fb_WormWeight(
	nLine:= 1, 
	UnitID:= 5, 
	fFast_Speed_vibrating_funnel:= fFast_Speed_vibrating_funnel, 
	fSlow_Speed_vibrating_funnel_1:= fSlow_Speed_vibrating_funnel_1, 
	fSlow_Speed_vibrating_funnel_2:= fSlow_Speed_vibrating_funnel_2, 
	fDerisedWeight_Worm:= fDerisedWeight_Worm, 
	fChangeMode_Worm_1:= fChangeMode_Worm_1, 
	fChangeMode_Worm_2:= fChangeMode_Worm_2, 
	fMaxWeight_Worm:= fMaxWeight_Worm, 
	fPerStop_Worm:= fPerStop_Worm, 
	fTimer_Worm:= fTimer_Worm, 
	fTimer_Alarm_Worm:= fTimer_Alarm_Worm, 
	fTimer_Check_Worm:= fTimer_Check_Worm, 
	fTimer_Check_Cylinder:= fTimer_Check_Cylinder, 
	fDelta_Worm:= fDelta_Worm,
	fTimer_Error_Worm:= fTimer_Error_Worm, 
	fProductLog=> fProductLog[2],
	bStatus_Worm=>bStatus_Worm,
	Time_start=>Time_Start_Worm_line1,
	Time_Stop=>Time_Stop_Worm_line1,
	status=>bStatus_Worm_line1,
	fweight_iot =>fWeight_Worm_line1);

IF bClear1 THEN
	nResult_false1 := 0;
	nResult_true1 := 0;
	nCount1 := 0;
	bClear1 := FALSE;
END_IF	

fDerisedWeight_Food_line1	:= fDerisedWeight_Food;
fDerisedWeight_Worm_line1	:= fDerisedWeight_Worm;
fActDelta_Food_line1		:= fb_FoodWeight.fActDelta_Food;
fActDelta_Worm_line1		:= fb_WormWeight.fActDelta_Worm;
fDelta_Food_line1			:= fb_FoodWeight.fDelta_Food;
fDelta_Worm_line1			:= fb_WormWeight.fDelta_Worm;
	
IF getuser = 'Operator' THEN
	bypassfood := FALSE;
	bypassWorm := FALSE;
END_IF

ACTION Auto:
CASE nState OF
	0:// int
		bStatus_Food_order[1] := FALSE;
		bStatus_Worm_order[1] := FALSE;
		bStatus_Lid_order[1]  := FALSE;
		fb_Transfer.Init();
		fb_FoodWeight.SetZero();
		fb_WormWeight.SetZero();
		nDoneTransferStop	  := 0;
		i1 		:= 0;
		i2 		:= 0;
		i3 		:= 0;
		bfinish1	:= TRUE;
		nState 	:= 1;
		
	1: // Start
		nState_FoodWeight := 0;
		nState_WormWeight := 0;
		nState_LidSupply := 0;
		nState_LidClose := 0;
		bResetAuto1			:= FALSE;
		bDoneCupSupply 		:= FALSE;
		bDoneFoodWeight 	:= FALSE;
		bDoneWormWeight 	:= FALSE;
		bDoneLidSupply 		:= FALSE;
		bDoneLidClose 		:= FALSE;
		fb_FoodWeight.SetZero();
		fb_WormWeight.SetZero();
		nState := 11;
	11:
		bResetAuto1			:= FALSE;
		nState_Dropcup := 0;
		nState_Transfer := 0;
		bStop1 := FALSE;
		bShift_is_over1 := FALSE;
		bStatusStart1 := FALSE;
		fb_FoodMixer.Stop();
		nStatus1	:= 'STOP';
		bFinishCupSupply 	:= FALSE;
		bFinishFoodWeight 	:= FALSE;
		bFinishWormWeight	:= FALSE;
		bFinishLidSupply	:= FALSE;
		bFinishLidClose		:= FALSE;
		bFinishTransfer		:= FALSE;
		bfinish1	:= TRUE;
		nState := 22;
	22:
		IF bStart1 THEN
			bfinish1		:= FALSE;
			bStatusStart1 	:= TRUE;
			bToDropcup1 	:= FALSE;
			bResetAuto1		:= TRUE;
			status			:= 'RUN';
			nState := 2;
		END_IF
		
	2: // start mode auto
		bfinish1		:= FALSE;
		nStatus1	:= 'RUN';
		bResetAuto1		:= TRUE;
		bStart1 := FALSE;
		IF bypassfood THEN
			fb_FoodMixer.Stop();
		ELSE
			fb_FoodMixer.Auto();
		END_IF
		fb_CupSupply.CheckCup();
		fb_LidSupply.CheckLid();
		bDone(CLK := bDoneTransfer);
		CASE nstateCycle OF 
			0:
				fbTimerCycle(IN := TRUE, PT := T#100S);
				IF bDone.Q THEN
					nstateCycle := 1;
				END_IF
			1:
				timeCycle := TIME_TO_REAL(fbTimerCycle.ET)/1000;
				nstateCycle := 2;
			2: 
				fproduct :=  REAL_TO_INT(3600/(timeCycle+0.001));
				fbTimerCycle(IN := FALSE);
				nstateCycle := 0;
		END_CASE
		CASE nState_Dropcup OF
			0:// waiting for transfer
				fbDelay(IN := FALSE);
				fb_CupSupply.HoldCup();
				IF bToDropcup1 THEN
					nState_Dropcup := 1;
				END_IF
			1:// dropcup
				IF fb_CupSupply.DropCup() THEN
					bDoneCupSupply := TRUE;
					bToDropcup1 := FALSE;
					nState_Dropcup := 2;
				END_IF
			2:
				fbDelay(IN := TRUE, PT := T#300MS);
				IF fbDelay.Q THEN
					nState_Dropcup := 0;
				END_IF
		END_CASE
		
		CASE nState_FoodWeight OF
			0:// waiting for transfer
				IF bDoneTransfer THEN
					i1 := i1 + 1;
					fbTimer(IN := FALSE);
					nState_FoodWeight := 1;	
				END_IF
			1:// Check cup present
				IF NOT fb_FoodWeight.bIsCupPresent THEN
					IF bypassfood THEN
						nState_FoodWeight := 3;
						bStatus_Food_order[i1] := TRUE;
					ELSE
						nState_FoodWeight := 2;
					END_IF
				ELSE
					bStatus_Food_order[i1] := FALSE;
					nState_FoodWeight := 3;
				END_IF
			2:// FoodWeight
				IF NOT fb_FoodWeight.bIsCupPresent THEN
					IF fb_FoodWeight.Auto() THEN
						bStatus_Food_order[i1] := bStatus_Food;
						nState_FoodWeight := 3;
					END_IF
				ELSE
					nState_FoodWeight := 22;
				END_IF 
			22:
				fbTimer(IN := TRUE, PT := T#0.3S);
				fb_FoodWeight.Auto();
				IF fbTimer.Q THEN
					fb_FoodWeight.Init();
					nState_FoodWeight := 0;
				END_IF
			3:// check i
				IF i1 < 3 THEN
					nState_FoodWeight := 5;
				ELSE 
					i1 := 2;
					nState_FoodWeight := 4;
				END_IF
			4:// dao vi tri
				bStatus_Food_order[1] := bStatus_Food_order[2];
				bStatus_Food_order[2] := bStatus_Food_order[3];
				nState_FoodWeight := 5;
			5:// Done
				bDoneFoodWeight := TRUE;
				nState_FoodWeight := 10;
		END_CASE
		
		CASE nState_WormWeight OF
			0: // waiting for transfer
				IF bDoneTransfer THEN
					i2 := i2 + 1;;
					fbTimer(IN := FALSE);
					nState_WormWeight := 1;
				END_IF
			1:
				IF NOT fb_WormWeight.bIsCupPresent THEN
					nCount1 := nCount1 + 1;
					nState_WormWeight := 11;
				ELSE
					bStatus_Worm_order[i2] := FALSE;
					nState_WormWeight := 3;
				END_IF
			11: // check food
				IF bStatus_Food_order[1] THEN
					IF bypassWorm THEN
						nState_WormWeight := 3;
						bStatus_Worm_order[i2] := TRUE;
					ELSE
						nState_WormWeight := 2;
					END_IF
				ELSE
					bStatus_Worm_order[i2] := FALSE;
					nState_WormWeight := 3;
				END_IF	
			2:// WormWeight
				IF NOT fb_WormWeight.bIsCupPresent THEN
					IF fb_WormWeight.Auto() THEN
						bStatus_Worm_order[i2] := bStatus_Worm;
						nState_WormWeight := 3;
					END_IF
				ELSE
					nState_WormWeight := 22;
				END_IF
			22:
				fbTimer(IN := TRUE, PT := T#0.3S);
				fb_WormWeight.Auto(); 
				IF fbTimer.Q THEN
					fb_WormWeight.Init();
					nState_WormWeight := 0;
				END_IF
			3:// check i
				IF bStatus_Worm_order[i2] THEN
					nResult_true1 := nResult_true1 + 1;
				END_IF
				IF i2 < 3 THEN
					nState_WormWeight := 5;
				ELSE
					i2 := 2;
					nState_WormWeight := 4;
				END_IF
			4:// dao vi tri
				nResult_false1 := nCount1 - nResult_true1;
				bStatus_Worm_order[1] := bStatus_Worm_order[2];
				bStatus_Worm_order[2] := bStatus_Worm_order[3];
				nState_WormWeight 	  := 5;
			5:// Done 
				bDoneWormWeight       := TRUE;
				nState_WormWeight	  := 10;
		END_CASE
		
		CASE nState_LidSupply OF
			0:// waiting for transfer
				IF bDoneTransfer THEN
					i3 := i3 + 1;
					nState_LidSupply := 1;
				END_IF
			1:// check worm
				IF bStatus_Worm_order[1] THEN
					IF bypassLid THEN
						bStatus_Lid_order[i3] := FALSE;
						nState_LidSupply := 4;
					ELSE
						nState_LidSupply := 2;
					END_IF
				ELSE
					bStatus_Lid_order[i3] := FALSE;
					nState_LidSupply := 4;
				END_IF
			2:// take lid
				IF fb_LidSupply.TakeLid() THEN
					nState_LidSupply := 3;
				END_IF
			3:// drop lid
				IF fb_LidSupply.DropLid() THEN
					bStatus_Lid_order[i3] := TRUE;
					nState_LidSupply := 4;
				END_IF
			4:// check i
				IF i3 < 3 THEN
					nState_LidSupply := 6;
				ELSE
					i3 := 2;
					nState_LidSupply := 5;
				END_IF
			5:// dao vi tri
				bStatus_Lid_order[1] := bStatus_Lid_order[2];
				bStatus_Lid_order[2] := bStatus_Lid_order[3];
				nState_LidSupply 	 := 6;
			6:// Done
				bDoneLidSupply 		 := TRUE;
				nState_LidSupply 	 := 10;
		END_CASE
		
		CASE nState_LidClose OF
			0: // waiting for transfer
				IF bDoneTransfer THEN
					nState_LidClose := 1;
				END_IF
			1:// Check lid supply
				IF  bStatus_Lid_order[1] THEN
					nState_LidClose := 2;
				ELSE
					nState_LidClose := 3;
				END_IF
			2:// Close lid
				IF fb_LidClose.CloseLid() THEN
					nState_LidClose := 3;
				END_IF
			3://Done
				bDoneLidClose := TRUE;
				nState_LidClose := 10;
		END_CASE
		
		CASE nState_Transfer OF
			0:// waiting for Done module
				IF nDoneTransfer = 0 THEN
					nState_Transfer := 1;
				ELSIF nDoneTransfer > 0 THEN
					IF bDoneCupSupply AND bDoneFoodWeight AND bDoneWormWeight AND bDoneLidSupply AND bDoneLidClose THEN
						nState_Transfer := 1;
					END_IF
				END_IF
			1:
				IF fb_CupSupply.isCupDrop THEN
					bDoneCupSupply 	:= FALSE;
					bDoneFoodWeight := FALSE;
					bDoneWormWeight := FALSE;
					bDoneLidSupply 	:= FALSE;
					bDoneLidClose 	:= FALSE;
					nState_Transfer := 11;
				ELSE 
					F_SetError(2,nLine:=1);
				END_IF
			11:// transfer
				IF fb_Transfer.Auto() THEN
					nShoot1 := nShoot1 + 1; 
					nState_Transfer:= 2;
				END_IF
			2:
				nState_FoodWeight := 0;
				nState_WormWeight := 0;
				nState_LidSupply  := 0;
				nState_LidClose	  := 0;
				nState_Transfer	  := 0;
		END_CASE
		//Stop button
		IF bStop1 THEN
			nState := 3;
			bStartLine1 := FALSE;
		ELSIF bShift_is_over1 THEN
			nState := 4;
		END_IF
	3://Stop
		bfinish1 := FALSE;
		fb_CupSupply.CheckCup();
		fb_LidSupply.CheckLid();
		bResetAuto1		:= TRUE;
		nStatus1	:= 'RUN';
		IF bypassfood THEN
			fb_FoodMixer.Stop();
		ELSE
			fb_FoodMixer.Auto();
		END_IF
		CASE nState_Dropcup OF
			0:// waiting for transfer
				fbDelay(IN := FALSE);
				fb_CupSupply.HoldCup();
				IF bToDropcup1 THEN
					nState_Dropcup := 1;
				END_IF
				IF bFinishTransfer THEN
					nState_Dropcup := 10;
				END_IF
			1:// dropcup
				IF fb_CupSupply.DropCup() THEN
					bDoneCupSupply := TRUE;
					bToDropcup1 := FALSE;
					nState_Dropcup := 2;
				END_IF
			2:
				fbDelay(IN := TRUE, PT := T#300MS);
				IF fbDelay.Q THEN
					nState_Dropcup := 10;
				END_IF
			10:// finish
				bDoneCupSupply := TRUE;
				bFinishCupSupply := TRUE;
		END_CASE
		
		CASE nState_FoodWeight OF
			0:// waiting for transfer
				IF bDoneTransfer THEN
					i1 := i1 + 1;
					fbTimer(IN := FALSE);
					nState_FoodWeight := 1;	
				END_IF
			1:// Check cup present
				IF NOT fb_FoodWeight.bIsCupPresent THEN
					IF bypassfood THEN
						nState_FoodWeight := 3;
						bStatus_Food_order[i1] := TRUE;
					ELSE
						nState_FoodWeight := 2;
					END_IF
				ELSE
					bStatus_Food_order[i1] := FALSE;
					nState_FoodWeight := 3;
				END_IF
			2:// FoodWeight
				IF NOT fb_FoodWeight.bIsCupPresent THEN
					IF fb_FoodWeight.Auto() THEN
						bStatus_Food_order[i1] := bStatus_Food;
						nState_FoodWeight := 3;
					END_IF
				ELSE
					nState_FoodWeight := 22;
				END_IF 
			22:
				fbTimer(IN := TRUE, PT := T#0.3S);
				fb_FoodWeight.Auto();
				IF fbTimer.Q THEN
					fb_FoodWeight.Init();
					nState_FoodWeight := 0;
				END_IF
			3:// check i
				IF i1 < 3 THEN
					nState_FoodWeight := 5;
				ELSE 
					i1 := 2;
					nState_FoodWeight := 4;
				END_IF
			4:// dao vi tri
				bStatus_Food_order[1] := bStatus_Food_order[2];
				bStatus_Food_order[2] := bStatus_Food_order[3];
				nState_FoodWeight := 5;
			5:// Done
				bDoneFoodWeight := TRUE;
				nState_FoodWeight := 10;
			10:// finish
				bFinishFoodWeight := TRUE;
		END_CASE
		
		CASE nState_WormWeight OF
			0: // waiting for transfer
				IF bDoneTransfer THEN
					i2 := i2 + 1;;
					fbTimer(IN := FALSE);
					nState_WormWeight := 1;
				END_IF
			1:
				IF NOT fb_WormWeight.bIsCupPresent THEN
					nCount1 := nCount1 + 1;
					nState_WormWeight := 11;
				ELSE
					bStatus_Worm_order[i2] := FALSE;
					nState_WormWeight := 3;
				END_IF
			11: // check food
				IF bStatus_Food_order[1] THEN
					IF bypassWorm THEN
						nState_WormWeight := 3;
						bStatus_Worm_order[i2] := TRUE;
					ELSE
						nState_WormWeight := 2;
					END_IF
				ELSE
					bStatus_Worm_order[i2] := FALSE;
					nState_WormWeight := 3;
				END_IF	
			2:// WormWeight
				IF NOT fb_WormWeight.bIsCupPresent THEN
					IF fb_WormWeight.Auto() THEN
						bStatus_Worm_order[i2] := bStatus_Worm;
						nState_WormWeight := 3;
					END_IF
				ELSE
					nState_WormWeight := 22;
				END_IF
			22:
				fbTimer(IN := TRUE, PT := T#0.3S);
				fb_WormWeight.Auto(); 
				IF fbTimer.Q THEN
					fb_WormWeight.Init();
					nState_WormWeight := 0;
				END_IF
			3:// check i
				IF bStatus_Worm_order[i2] THEN
					nResult_true1 := nResult_true1 + 1;
				END_IF
				IF i2 < 3 THEN
					nState_WormWeight := 5;
				ELSE
					i2 := 2;
					nState_WormWeight := 4;
				END_IF
			4:// dao vi tri
				nResult_false1 := nCount1 - nResult_true1;
				bStatus_Worm_order[1] := bStatus_Worm_order[2];
				bStatus_Worm_order[2] := bStatus_Worm_order[3];
				nState_WormWeight 	  := 5;
			5:// Done 
				bDoneWormWeight       := TRUE;
				nState_WormWeight	  := 10;
			10:// finish
				bFinishWormWeight	  := TRUE;
		END_CASE
		
		CASE nState_LidSupply OF
			0:// waiting for transfer
				IF bDoneTransfer THEN
					i3 := i3 + 1;
					nState_LidSupply := 1;
				END_IF
			1:// check worm
				IF bStatus_Worm_order[1] THEN
					IF bypassLid THEN
						bStatus_Lid_order[i3] := FALSE;
						nState_LidSupply := 4;
					ELSE
						nState_LidSupply := 2;
					END_IF
				ELSE
					bStatus_Lid_order[i3] := FALSE;
					nState_LidSupply := 4;
				END_IF
			2:// take lid
				IF fb_LidSupply.TakeLid() THEN
					nState_LidSupply := 3;
				END_IF
			3:// drop lid
				IF fb_LidSupply.DropLid() THEN
					bStatus_Lid_order[i3] := TRUE;
					nState_LidSupply := 4;
				END_IF
			4:// check i
				IF i3 < 3 THEN
					nState_LidSupply := 6;
				ELSE
					i3 := 2;
					nState_LidSupply := 5;
				END_IF
			5:// dao vi tri
				bStatus_Lid_order[1] := bStatus_Lid_order[2];
				bStatus_Lid_order[2] := bStatus_Lid_order[3];
				nState_LidSupply 	 := 6;
			6:// Done
				bDoneLidSupply 		 := TRUE;
				nState_LidSupply 	 := 10;
			10:// finish
				bFinishLidSupply	 := TRUE;
		END_CASE
		
		CASE nState_LidClose OF
			0: // waiting for transfer
				IF bDoneTransfer THEN
					nState_LidClose := 1;
				END_IF
			1:// Check lid supply
				IF  bStatus_Lid_order[1] THEN
					nState_LidClose := 2;
				ELSE
					nState_LidClose := 3;
				END_IF
			2:// Close lid
				IF fb_LidClose.CloseLid() THEN
					nState_LidClose := 3;
				END_IF
			3://Done
				bDoneLidClose   := TRUE;
				nState_LidClose := 10;
			10:// finish
				bFinishLidClose := TRUE;
		END_CASE
		
		CASE nState_Transfer OF
			0:// waiting for Done module
				IF nDoneTransfer = 0 THEN
					nState_Transfer := 10;
				ELSIF nDoneTransfer > 0 THEN
					IF bDoneCupSupply AND bDoneFoodWeight AND bDoneWormWeight AND bDoneLidSupply AND bDoneLidClose THEN
					nState_Transfer := 10;
					END_IF
				END_IF
			1:
				IF fb_CupSupply.isCupDrop THEN
					bDoneCupSupply 	:= FALSE;
					bDoneFoodWeight := FALSE;
					bDoneWormWeight := FALSE;
					bDoneLidSupply 	:= FALSE;
					bDoneLidClose 	:= FALSE;
					nState_Transfer := 11;
				ELSE 
					F_SetError(2,nLine:=1);
				END_IF
			11:// transfer
				IF fb_Transfer.Auto() THEN
					nShoot1 := nShoot1 + 1;
					nState_Transfer:= 2;
				END_IF
			2: 
				nState_FoodWeight := 0;
				nState_WormWeight := 0;
				nState_LidSupply  := 0;
				nState_LidClose	  := 0;
				nState_Dropcup 	  := 0;
				nState_Transfer   := 0;
			10:// finish
				bFinishTransfer		:= TRUE;	
		END_CASE
		
		IF bFinishCupSupply AND bFinishFoodWeight AND bFinishWormWeight AND bFinishLidSupply AND bFinishLidClose AND bFinishTransfer THEN
			bfinish1	:= TRUE;
			nState := 11;
		END_IF
	4:// shift is over
		bfinish1 := FALSE;
		bStart1	:= FALSE;
		IF bypassfood THEN
			fb_FoodMixer.Stop();
		ELSE
			fb_FoodMixer.Auto();
		END_IF
		fb_CupSupply.CheckCup();
		fb_LidSupply.CheckLid();
		bResetAuto1		:= TRUE;
		bStatusStart1 := FALSE;
		nStatus1	:= 'RUN';
		bDone(CLK := bDoneTransfer);
		CASE nstateCycle OF 
			0:
				fbTimerCycle(IN := TRUE, PT := T#30S);
				IF bDone.Q THEN
					nstateCycle := 1;
				END_IF
			1:
				timeCycle := TIME_TO_REAL(fbTimerCycle.ET)/1000;
				nstateCycle := 2;
			2: 
				fproduct  := REAL_TO_INT(3600/(timeCycle+0.001));
				fbTimerCycle(IN := FALSE);
				nstateCycle := 0;
		END_CASE
		
		CASE nState_Dropcup OF
			0:// waiting for transfer
				fbDelay(IN := FALSE);
				fb_CupSupply.HoldCup();
				IF bToDropcup1 THEN
					nState_Dropcup := 10;
				END_IF
			1:// dropcup
				IF fb_CupSupply.DropCup() THEN
					bDoneCupSupply := TRUE;
					bToDropcup1 := FALSE;
					nState_Dropcup := 2;
				END_IF
			2:
				fbDelay(IN := TRUE, PT := T#300MS);
				IF fbDelay.Q THEN
					nState_Dropcup := 10;
				END_IF
			10:// finish
				bDoneCupSupply := TRUE;
				bFinishCupSupply := TRUE;
		END_CASE
		
		CASE nState_FoodWeight OF
			0:// waiting for transfer
				IF bDoneTransfer AND nDoneTransferStop < 4 THEN
					i1 := i1 + 1;
					fbTimer(IN := FALSE);
					nState_FoodWeight := 1;	
				ELSIF bDoneTransfer AND nDoneTransferStop >= 4 THEN
					i1 := i1 + 1;
					fbTimer(IN := FALSE);
					nState_FoodWeight := 33;	
				END_IF
			1:// Check cup present
				IF NOT fb_FoodWeight.bIsCupPresent THEN
					IF bypassfood THEN
						nState_FoodWeight := 3;
						bStatus_Food_order[i1] := TRUE;
					ELSE
						nState_FoodWeight := 2;
					END_IF
				ELSE
					bStatus_Food_order[i1] := FALSE;
					nState_FoodWeight := 3;
				END_IF
			2:// FoodWeight
				IF NOT fb_FoodWeight.bIsCupPresent THEN
					IF fb_FoodWeight.Auto() THEN
						bStatus_Food_order[i1] := bStatus_Food;
						nState_FoodWeight := 3;
					END_IF
				ELSE
					nState_FoodWeight := 22;
				END_IF 
			22:
				fbTimer(IN := TRUE, PT := T#0.3S);
				fb_FoodWeight.Auto();
				IF fbTimer.Q THEN
					fb_FoodWeight.Init();
					nState_FoodWeight := 0;
				END_IF
			33:
				bStatus_Food_order[i1] := FALSE;
				nState_FoodWeight := 3;
			3:// check i
				IF i1 < 3 THEN
					nState_FoodWeight := 5;
				ELSE 
					i1 := 2;
					nState_FoodWeight := 4;
				END_IF
			4:// dao vi tri
				bStatus_Food_order[1] := bStatus_Food_order[2];
				bStatus_Food_order[2] := bStatus_Food_order[3];
				nState_FoodWeight := 5;
			5:// Done
				bDoneFoodWeight := TRUE;
				nState_FoodWeight := 10;
			10:// finish
				bFinishFoodWeight := TRUE;
		END_CASE
		
		CASE nState_WormWeight OF
			0: // waiting for transfer
				IF bDoneTransfer AND nDoneTransferStop < 6 THEN
					i2 := i2 + 1;;
					fbTimer(IN := FALSE);
					nState_WormWeight := 1;
				ELSIF bDoneTransfer AND nDoneTransferStop >= 6 THEN
					i2 := i2 + 1;;
					fbTimer(IN := FALSE);
					nState_WormWeight := 33;
				END_IF
			1:
				IF NOT fb_WormWeight.bIsCupPresent THEN
					nCount1 := nCount1 + 1;
					nState_WormWeight := 11;
				ELSE
					bStatus_Worm_order[i2] := FALSE;
					nState_WormWeight := 3;
				END_IF
			11: // check food
				IF bStatus_Food_order[1] THEN
					IF bypassWorm THEN
						nState_WormWeight := 3;
						bStatus_Worm_order[i2] := TRUE;
					ELSE
						nState_WormWeight := 2;
					END_IF
				ELSE
					bStatus_Worm_order[i2] := FALSE;
					nState_WormWeight := 3;
				END_IF	
			2:// WormWeight
				IF NOT fb_WormWeight.bIsCupPresent THEN
					IF fb_WormWeight.Auto() THEN
						bStatus_Worm_order[i2] := bStatus_Worm;
						nState_WormWeight := 3;
					END_IF
				ELSE
					nState_WormWeight := 22;
				END_IF
			22:
				fbTimer(IN := TRUE, PT := T#0.3S);
				fb_WormWeight.Auto(); 
				IF fbTimer.Q THEN
					fb_WormWeight.Init();
					nState_WormWeight := 0;
				END_IF
			33:
				bStatus_Worm_order[i2] := FALSE;
				nState_WormWeight := 3;
			3:// check i
				IF bStatus_Worm_order[i2] THEN
					nResult_true1 := nResult_true1 + 1;
				END_IF
				IF i2 < 3 THEN
					nState_WormWeight := 5;
				ELSE
					i2 := 2;
					nState_WormWeight := 4;
				END_IF
			4:// dao vi tri
				nResult_false1 := nCount1 - nResult_true1;
				bStatus_Worm_order[1] := bStatus_Worm_order[2];
				bStatus_Worm_order[2] := bStatus_Worm_order[3];
				nState_WormWeight 	  := 5;
			5:// Done 
				bDoneWormWeight       := TRUE;
				nState_WormWeight	  := 10;
			10:// finish
				bFinishWormWeight	  := TRUE;
		END_CASE
		
		CASE nState_LidSupply OF
			0:// waiting for transfer
				IF bDoneTransfer THEN
					i3 := i3 + 1;
					nState_LidSupply := 1;
				END_IF
			1:// check worm
				IF bStatus_Worm_order[1] THEN
					IF bypassLid THEN
						bStatus_Lid_order[i3] := FALSE;
						nState_LidSupply := 4;
					ELSE
						nState_LidSupply := 2;
					END_IF
				ELSE
					bStatus_Lid_order[i3] := FALSE;
					nState_LidSupply := 4;
				END_IF
			2:// take lid
				IF fb_LidSupply.TakeLid() THEN
					nState_LidSupply := 3;
				END_IF
			3:// drop lid
				IF fb_LidSupply.DropLid() THEN
					bStatus_Lid_order[i3] := TRUE;
					nState_LidSupply := 4;
				END_IF
			4:// check i
				IF i3 < 3 THEN
					nState_LidSupply := 6;
				ELSE
					i3 := 2;
					nState_LidSupply := 5;
				END_IF
			5:// dao vi tri
				bStatus_Lid_order[1] := bStatus_Lid_order[2];
				bStatus_Lid_order[2] := bStatus_Lid_order[3];
				nState_LidSupply 	 := 6;
			6:// Done
				bDoneLidSupply 		 := TRUE;
				nState_LidSupply 	 := 10;
			10:// finish
				bFinishLidSupply	 := TRUE;
		END_CASE
		
		CASE nState_LidClose OF
			0: // waiting for transfer
				IF bDoneTransfer THEN
					nState_LidClose := 1;
				END_IF
			1:// Check lid supply
				IF  bStatus_Lid_order[1] THEN
					nState_LidClose := 2;
				ELSE
					nState_LidClose := 3;
				END_IF
			2:// Close lid
				IF fb_LidClose.CloseLid() THEN
					nState_LidClose := 3;
				END_IF
			3://Done
				bDoneLidClose   := TRUE;
				nState_LidClose := 10;
			10:// finish
				bFinishLidClose := TRUE;
		END_CASE
		
		CASE nState_Transfer OF
			0:// waiting for Done module
				IF bDoneCupSupply AND bDoneFoodWeight AND bDoneWormWeight AND bDoneLidSupply AND bDoneLidClose THEN
					nState_Transfer := 1;
				END_IF
			1:
				IF fb_CupSupply.isCupDrop THEN
					bDoneCupSupply 	:= FALSE;
					bDoneFoodWeight := FALSE;
					bDoneWormWeight := FALSE;
					bDoneLidSupply 	:= FALSE;
					bDoneLidClose 	:= FALSE;
					nState_Transfer := 11;
				ELSE 
					F_SetError(2,nLine:=1);
				END_IF
			11:// transfer
				IF fb_Transfer.Auto() THEN
					nShoot1 := nShoot1 + 1;
					nState_Transfer:= 2;
				END_IF
			2:
				nState_FoodWeight := 0;
				nState_WormWeight := 0;
				nState_LidSupply  := 0;
				nState_LidClose	  := 0;
				nDoneTransferStop := nDoneTransferStop + 1;
				nState_Transfer   := 3;
			3:
				IF nDoneTransferStop < 11 THEN
					nState_Transfer   := 0;
				ELSE
					nState_Transfer   := 10;
				END_IF
			10:// finish
				bFinishTransfer		:= TRUE;
		END_CASE
		IF bFinishCupSupply AND bFinishFoodWeight AND bFinishWormWeight AND bFinishLidSupply AND bFinishLidClose AND bFinishTransfer THEN
			bfinish1	:= TRUE;
			nState := 0;
		END_IF
END_CASE
END_ACTION

ACTION check:
IF fb_CupSupply.fbCylinder_Up.bIsRetract THEN
	bCylinder_up_retract 	:= TRUE;
	bCylinder_up_extend		:= FALSE;
ELSE
	bCylinder_up_retract 	:= FALSE;
	bCylinder_up_extend		:= TRUE;
END_IF

IF fb_CupSupply.fbCylinder_Dw.bIsExtend THEN
	bCylinder_dw_extend 	:= TRUE;
	bCylinder_dw_retract 	:= FALSE;
ELSIF fb_CupSupply.fbCylinder_Dw.bIsRetract THEN
	bCylinder_dw_extend 	:= FALSE;
	bCylinder_dw_retract 	:= TRUE;
ELSE
	bCylinder_dw_extend 	:= FALSE;
	bCylinder_dw_retract 	:= FALSE;
END_IF

IF fb_CupSupply.fbCylinder_Suction.bIsExtend THEN
	bCylinder_Suction_cup_extend 	:= TRUE;
	bCylinder_Suction_cup_retract	:= FALSE;
ELSE
	bCylinder_Suction_cup_extend 	:= FALSE;
	bCylinder_Suction_cup_retract	:= TRUE;
END_IF
//--------------------------------------
IF fb_WormWeight.fbCylinder.bIsRetract THEN
	bCylinder_Block_Worm_Extend	 := FALSE;
	bCylinder_Block_Worm_Retract := TRUE;
ELSE
	bCylinder_Block_Worm_Extend	 := TRUE;
	bCylinder_Block_Worm_Retract := FALSE;
END_IF
//--------------------------------------
IF fb_LidSupply.fbCylinder_LidStopper.bIsExtend THEN
	bCylinder_LidStopper_extend 	:= TRUE;
	bCylinder_LidStopper_retract 	:= FALSE;
ELSIF fb_LidSupply.fbCylinder_LidStopper.bIsRetract THEN
	bCylinder_LidStopper_extend 	:= FALSE;
	bCylinder_LidStopper_retract 	:= TRUE;
ELSE
	bCylinder_LidStopper_extend 	:= FALSE;
	bCylinder_LidStopper_retract 	:= FALSE;
END_IF

IF fb_LidSupply.fbCylinder_Suction.bIsExtend THEN
	bCylinder_Suction_extend		:= TRUE;
	bCylinder_Suction_retract		:= FALSE;
ELSIF fb_LidSupply.fbCylinder_Suction.bIsRetract THEN
	bCylinder_Suction_extend		:= FALSE;
	bCylinder_Suction_retract		:= TRUE;
ELSE
	bCylinder_Suction_extend		:= FALSE;
	bCylinder_Suction_retract		:= FALSE;
END_IF
//--------------------------------------
IF fb_LidClose.fbCylinder_LidClose.bIsExtend THEN
	bCylinder_CloseLid_Extend		:= TRUE;
	bCylinder_CloseLid_Retract		:= FALSE;
ELSIF fb_LidClose.fbCylinder_LidClose.bIsRetract THEN
	bCylinder_CloseLid_Extend		:= FALSE;
	bCylinder_CloseLid_Retract		:= TRUE;
ELSE
	bCylinder_CloseLid_Extend		:= FALSE;
	bCylinder_CloseLid_Retract		:= FALSE;
END_IF
//--------------------------------------
IF fb_Transfer.fbCylinder_Comb.bIsExtend THEN
	bCylinder_Comb_Extend			:= TRUE;
	bCylinder_Comb_Retract			:= FALSE;
ELSIF fb_Transfer.fbCylinder_Comb.bIsRetract THEN
	bCylinder_Comb_Extend			:= FALSE;
	bCylinder_Comb_Retract			:= TRUE;
ELSE
	bCylinder_Comb_Extend			:= FALSE;
	bCylinder_Comb_Retract			:= FALSE;
END_IF

IF fb_Transfer.fbCylinder_Clip.bIsExtend THEN
	bCylinder_Clip_Extend			:= TRUE;
	bCylinder_Clip_Retract			:= FALSE;
ELSIF fb_Transfer.fbCylinder_Clip.bIsRetract THEN
	bCylinder_Clip_Extend			:= FALSE;
	bCylinder_Clip_Retract			:= TRUE;
ELSE
	bCylinder_Clip_Extend			:= FALSE;
	bCylinder_Clip_Retract			:= FALSE;
END_IF

IF fb_Transfer.fbCylinder_Move_Comb.bIsExtend THEN
	bCylinder_Move_Comb_Extend		:= TRUE;
	bCylinder_Move_Comb_Retract		:= FALSE;
ELSIF fb_Transfer.fbCylinder_Move_Comb.bIsRetract THEN
	bCylinder_Move_Comb_Extend		:= FALSE;
	bCylinder_Move_Comb_Retract		:= TRUE;
ELSE
	bCylinder_Move_Comb_Extend		:= FALSE;
	bCylinder_Move_Comb_Retract		:= FALSE;
END_IF

bMotor_mixer_Manual				:= FALSE;
bMotor_mixer_reverse			:= FALSE;
bMotor_Food						:= FALSE;
bMotor_Food_reverse				:= FALSE;
bMotor_vibrating_funnel			:= FALSE;
END_ACTION

ACTION Check_reset:
IF fb_CupSupply.fbCylinder_Up.bIsRetract AND fb_CupSupply.fbCylinder_Dw.bIsExtend 
	AND NOT fb_WormWeight.fbCylinder.bIsRetract AND fb_LidSupply.fbCylinder_Suction.bIsRetract 
	AND fb_LidClose.fbCylinder_LidClose.bIsRetract AND fb_Transfer.fbCylinder_Comb.bIsRetract 
	AND fb_Transfer.fbCylinder_Clip.bIsRetract AND fb_Transfer.fbCylinder_Move_Comb.bIsRetract
	AND fb_CupSupply.fbCylinder_Suction.bIsExtend THEN
		bResetmanual1 := TRUE;
ELSE 
		bResetmanual1 := FALSE;
END_IF
IF bReset THEN
	bCylinder_up_retract 	:= TRUE;
	bCylinder_up_extend		:= FALSE;
	bCylinder_dw_extend 	:= TRUE;
	bCylinder_dw_retract 	:= FALSE;
	bCylinder_Suction_cup_retract 	:= FALSE;
	bCylinder_Suction_cup_extend 	:= TRUE;
	bCylinder_Block_Worm_Extend	 := TRUE;
	bCylinder_Block_Worm_Retract := FALSE;
	bCylinder_Suction_extend		:= FALSE;
	bCylinder_Suction_retract		:= TRUE;
	bCylinder_CloseLid_Extend		:= FALSE;
	bCylinder_CloseLid_Retract		:= TRUE;
	bCylinder_Comb_Extend			:= FALSE;
	bCylinder_Comb_Retract			:= TRUE;
	bCylinder_Clip_Extend			:= FALSE;
	bCylinder_Clip_Retract			:= TRUE;
	IF fb_Transfer.fbCylinder_Comb.bIsRetract THEN
		bCylinder_Move_Comb_Extend		:= FALSE;
		bCylinder_Move_Comb_Retract		:= TRUE;
	END_IF
	bxa := FALSE;
END_IF
END_ACTION

ACTION Init:
fb_CupSupply.Init();
fb_FoodWeight.Init();
fb_WormWeight.Init();
fb_LidSupply.Init();
fb_LidClose.Init();
fb_Transfer.Init();

nState := 0;
nState_Dropcup := 0;
nState_FoodWeight := 0;
nState_WormWeight := 0;
nState_LidSupply := 0;
nState_LidClose := 0;
nState_Transfer := 0;

bFinishCupSupply 	:= FALSE;
bFinishFoodWeight 	:= FALSE;
bFinishWormWeight	:= FALSE;
bFinishLidSupply	:= FALSE;
bFinishLidClose		:= FALSE;
bFinishTransfer		:= FALSE;

bDoneCupSupply 		:= FALSE;
bDoneFoodWeight 	:= FALSE;
bDoneWormWeight 	:= FALSE;
bDoneLidSupply 		:= FALSE;
bDoneLidClose 		:= FALSE;
bDoneTransfer		:= FALSE;
nDoneTransferStop	  := 0;

bStatus_Food_order[1] := FALSE;
bStatus_Worm_order[1] := FALSE;
bStatus_Lid_order[1]  := FALSE;
		
i1 		:= 0;
i2 		:= 0;
i3 		:= 0;
END_ACTION

ACTION Manual:
fb_CupSupply.Manual(bCylinder_dw_extend := bCylinder_dw_extend, bCylinder_dw_retract := bCylinder_dw_retract,
					bCylinder_up_extend := bCylinder_up_extend, bCylinder_up_retract := bCylinder_up_retract,
					bCylinder_suction_extend:= bCylinder_Suction_cup_extend, bCylinder_suction_retract := bCylinder_Suction_cup_retract);

IF bxa THEN
	IF daothucan THEN
		fb_FoodMixer.Auto();
	ELSE
		fb_FoodMixer.Stop();
	END_IF
ELSE
	daothucan := FALSE;	
	fb_FoodMixer.Manual(bDown_Motor_Mixer := bDown_Motor_Mixer, bUp_Motor_Mixer := bUp_Motor_Mixer,
					bMotor_mixer_Manual := bMotor_mixer_Manual,bMotor_mixer_reverse := bMotor_mixer_reverse);

	IF bUp_Motor_Mixer THEN
		bUp_Motor_Mixer := FALSE;
	END_IF
	
	IF bDown_Motor_Mixer THEN
		bDown_Motor_Mixer := FALSE;
	END_IF
END_IF

IF bxa THEN
	CASE nstatetest1 OF 
	0:
		IF xathucan THEN
			nstatetest1 := 1;			
		END_IF
	1:
		IF fb_FoodWeight.Auto() THEN
			nstatetest1 := 2;
		END_IF
	2: 
		xathucan := FALSE;
		nstatetest1 := 3;
	3:
		nstatetest1 := 0;
	END_CASE
ELSE
	xathucan := FALSE;
	nstatetest1 := 0;
	fb_FoodWeight.Manual(bDown_Food_Motor := bDown_Food_Motor, bUp_Food_Motor := bUp_Food_Motor,
									bMotor_Food := bMotor_Food, bZero_Loadcell_Food := bZero_Loadcell_Food, bMotor_Food_Reverse := bMotor_Food_reverse);
				
	IF bUp_Food_Motor THEN
		bUp_Food_Motor := FALSE;
	END_IF
				
	IF bDown_Food_Motor THEN
		bDown_Food_Motor := FALSE;
	END_IF
				
	IF bZero_Loadcell_Food THEN
		bZero_Loadcell_Food := FALSE;
	END_IF
END_IF

IF bxa THEN
	CASE nstatetest2 OF 
	0:
		IF xasau THEN
			nstatetest2 := 1;
		END_IF
	1:
		IF fb_WormWeight.Auto() THEN
			nstatetest2 := 2;
		END_IF
	2: 
		xasau := FALSE;
		nstatetest2 := 3;
	3:
		nstatetest2 := 0;
	END_CASE
ELSE
	xasau := FALSE;
	nstatetest2 := 0;
	fb_WormWeight.Manual(bCylinder_Block_Worm_Extend := bCylinder_Block_Worm_Extend, bCylinder_Block_Worm_Retract := bCylinder_Block_Worm_Retract,
					bDown_vibrating_funnel := bDown_vibrating_funnel, bUp_vibrating_funnel := bUp_vibrating_funnel,
					bMotor_vibrating_funnel := bMotor_vibrating_funnel, bZero_Loadcell_Worm := bZero_Loadcell_Worm);
	
	IF bUp_vibrating_funnel THEN
		bUp_vibrating_funnel := FALSE;
	END_IF
	
	IF bDown_vibrating_funnel THEN
		bDown_vibrating_funnel := FALSE;
	END_IF
	
	IF bZero_Loadcell_Worm THEN
		bZero_Loadcell_Worm := FALSE;
	END_IF
END_IF

fb_LidSupply.Manual(bCylinder_LidStopper_extend := bCylinder_LidStopper_extend, bCylinder_LidStopper_retract := bCylinder_LidStopper_retract,
					bCylinder_Suction_extend := bCylinder_Suction_extend, bCylinder_Suction_retract := bCylinder_Suction_retract,
					bCupSuctionValve := bCupSuctionValve, bLidSuctionValve := bLidSuctionValve, bBlowValve := bBlowValve);

fb_LidClose.Manual(bCylinder_CloseLid_Extend := bCylinder_CloseLid_Extend, bCylinder_CloseLid_Retract := bCylinder_CloseLid_Retract);



fb_Transfer.Manual(bCylinder_Clip_Extend := bCylinder_Clip_Extend, bCylinder_Clip_Retract := bCylinder_Clip_Retract,
				   bCylinder_Comb_Extend := bCylinder_Comb_Extend, bCylinder_Comb_Retract := bCylinder_Comb_Retract,
				   bCylinder_Move_Comb_Extend := bCylinder_Move_Comb_Extend, bCylinder_Move_Comb_Retract := bCylinder_Move_Comb_Retract);

IF fb_CupSupply.fbCylinder_Suction.bIsExtend AND fb_LidSupply.fbCylinder_Suction.bIsRetract AND fb_LidClose.fbCylinder_LidClose.bIsRetract THEN
	bCheck := TRUE;
ELSE
	bCheck := FALSE;
END_IF
END_ACTION

ACTION Reset:
fb_CupSupply.Reset();
fb_FoodMixer.Reset();
fb_FoodWeight.Reset();
fb_WormWeight.Reset();
fb_LidSupply.Reset();
fb_LidClose.Reset();
fb_Transfer.Reset();
nState := 22;
END_ACTION

ACTION Stop:
fb_FoodWeight.Stop();
fb_WormWeight.Stop();
fb_LidSupply.Stop();
fb_LidClose.Stop();
fb_Transfer.Stop();
fb_CupSupply.Stop();
bLidSuctionValve		:= FALSE;
bCupSuctionValve		:= FALSE;
bResetAuto1				:= FALSE;
fb_FoodMixer.Stop();
END_ACTION

END_PROGRAM

// ---- POUs/Modules/FB_CupSupplyModule.TcPOU
FUNCTION_BLOCK FB_CupSupplyModule
VAR_INPUT
	nLine						: INT;
	timerCheckCylinder_Up		: REAL := 10;
	timerCheckCylinder_Dw		: REAL := 10;
	timerCylinder_Up_extend		: REAL;
	timerCylinder_Suction		: REAL;
	timerCylinder_Suction_extend: REAL;
	timerCheckEmpty				: REAL := 10;
	timerCheckStuck				: REAL := 10;
	ttimerCylinder_val			: REAL;
	timerCylinder_Suction_pick	: REAL;
END_VAR
VAR_OUTPUT
END_VAR
VAR
	// ===== CHILD COMPONENTS ======
	fbCylinder_Up				: FB_Cylinder;
	fbCylinder_Dw				: FB_Cylinder;
	fbCylinder_Suction			: FB_Cylinder;
	// ===== SIM COMPONENTS ======
	fbCylinderSim_Up			: FB_Cylinder_Sim;
	fbCylinderSim_Dw			: FB_Cylinder_Sim;
	fbCylinderSim_Suction		: FB_Cylinder_Sim;
	// ===== INTERFACES ======
	iCylinder_Up				: I_Cylinder;
	iCylinder_Dw				: I_Cylinder;
	iCylinder_Suction			: I_Cylinder;
	//===== Var IO ======
	bCupEmpty AT %I*			: BOOL;
	bCupDrop  AT %I*			: BOOL;
	//===== Var Auto ====
	//===== Var method
	nState_DropCup				: INT;
	nState_Enable				: INT;
	nState_Check				: INT;
	nState_siren				: INT;
	nState_Reset				: INT;
	tTimer_Enable1				: TON;
	tTimer_Enable2				: TON;
	tTimer_DropCup				: TON;
	tTimer_CheckCup				: TON;
	tTimer_Suction				: TON;
	tTimer_Up					: ton;
	tTimer_Dw					: TON;
	tTimer_Reset				: TON;
END_VAR

IF bSimMode THEN
	iCylinder_Up := fbCylinderSim_Up;
	fbCylinderSim_Up();
	iCylinder_Dw := fbCylinderSim_Dw;
	fbCylinderSim_Dw();
	iCylinder_Suction := fbCylinderSim_Suction;
	fbCylinderSim_Suction();
ELSE
	iCylinder_Up := fbCylinder_Up;
	fbCylinder_Up(id := 1);
	iCylinder_Dw := fbCylinder_Dw;
	fbCylinder_Dw(id := 1);
	iCylinder_Suction := fbCylinder_Suction;
	fbCylinder_Suction(id := 1);
END_IF

METHOD CheckCup : BOOL
VAR_INPUT
END_VAR
IF NOT isCupEmpty THEN
	CASE nState_Check OF
		0:
			IF nLine = 1 THEN
				F_SetWarning(101,nLine := 1);
			ELSIF nLine = 2 THEN
				F_SetWarning(108,nLine := 2);
			END_IF
			nState_Check := 1;
		1: 
			tTimer_CheckCup(IN := TRUE, PT := REAL_TO_TIME(timerCheckEmpty)*1000);
			IF tTimer_CheckCup.Q THEN
				IF nLine = 1 THEN
						F_SetError(1,nLine := 1);
				ELSIF nLine = 2 THEN
						F_SetError(23,nLine := 2);
				END_IF
			END_IF
	END_CASE
ELSE
	tTimer_CheckCup(IN := FALSE);
	nState_Check := 0;
END_IF

CASE nState_siren OF
	0:
		IF NOT isCupEmpty THEN
			nState_siren := 1;
		END_IF
	1:
		IF isCupEmpty THEN
			IF nLine = 1 THEN
				bWrn := FALSE;
			ELSIF nLine = 2 THEN
				bWrn2 := FALSE;
			END_IF
			bSirens := FALSE;
			nState_siren := 0;
		END_IF
END_CASE
END_METHOD

METHOD DropCup : BOOL
VAR_INPUT
END_VAR
CASE nState_DropCup OF
	0: //init
		DropCup := FALSE;
		tTimer_DropCup(IN := FALSE);
		tTimer_Suction(IN := FALSE);
		nState_DropCup := 1;
	1: //check CupEmpty
		nState_DropCup := 2;
	2: //cylinder_up extend to hold cup
		iCylinder_Up.Extend();
		iCylinder_Suction.Retract();
		tTimer_Suction(IN := TRUE, PT := REAL_TO_TIME(timerCylinder_Suction_extend)*1000);
		tTimer_DropCup(IN := TRUE, PT := REAL_TO_TIME(timerCylinder_Up_extend)*1000);
		IF tTimer_DropCup.Q AND tTimer_Suction.Q THEN
			nState_DropCup := 3;
		END_IF
	3: // cylinder_dw retract to dropcup
		iCylinder_Up.Extend();
		tTimer_Suction(IN := FALSE);
		tTimer_DropCup(IN := FALSE);
		iCylinder_Dw.Retract();
		nState_DropCup := 33;
	33:
		iCylinder_Up.Extend();
		iCylinder_Dw.Retract();
		iCylinder_Suction.Retract();
		tTimer_DropCup(IN := TRUE, PT := REAL_TO_TIME(timerCheckCylinder_Dw)*1000);
		IF tTimer_DropCup.Q THEN
			IF nLine = 1 THEN
				F_SetError(4,nLine := 1);
			ELSIF nLine = 2 THEN
				F_SetError(26,nLine := 2);
			END_IF
		ELSIF iCylinder_Dw.bIsRetract THEN
			tTimer_DropCup(IN := FALSE);
			nState_DropCup := 34;
		END_IF
	34:
		tTimer_DropCup(IN := TRUE, PT := REAL_TO_TIME(timerCylinder_Suction_pick)*1000);
		IF tTimer_DropCup.Q THEN
			nState_DropCup := 44;
		END_IF
	44:
		tTimer_DropCup(IN := FALSE);
		nState_DropCup := 4;
	4: // check not isCupDrop
		iCylinder_Up.Extend();
		iCylinder_Dw.Retract();
		iCylinder_Suction.Extend();
		tTimer_Suction(IN := TRUE, PT := REAL_TO_TIME(timerCylinder_Suction)*1000);
		IF NOT isCupDrop THEN //sensor NC
			tTimer_DropCup(IN := FALSE);
			nState_DropCup := 5;
		ELSE
			tTimer_DropCup(IN := TRUE, PT := REAL_TO_TIME(timerCheckStuck)*1000);
			IF tTimer_DropCup.Q THEN
				IF nLine = 1 THEN
					F_SetError(2,nLine := 1);
					nState_DropCup := 5;
				ELSIF nLine = 2 THEN
					F_SetError(24,nLine := 2);
					nState_DropCup := 5;
				END_IF
			END_IF
		END_IF
	5:
		tTimer_Dw(IN := TRUE, PT := REAL_TO_TIME(ttimerCylinder_val)*1000);
		IF tTimer_Dw.Q THEN
			iCylinder_Dw.Extend();
		END_IF
		IF iCylinder_Suction.bIsExtend THEN
			tTimer_Suction(IN := FALSE);
			nState_DropCup := 55;
		ELSE
			tTimer_Suction(IN := TRUE, PT := REAL_TO_TIME(timerCylinder_Suction)*1000);
			IF tTimer_Suction.Q THEN
				IF nLine = 1 THEN
					F_SetError(60,nLine := 1);
				ELSIF nLine = 2 THEN
					F_SetError(61,nLine := 2);
				END_IF
			END_IF
		END_IF
	55:
		tTimer_Dw(IN := false);
		IF isCupDrop THEN
			tTimer_DropCup(IN := FALSE);
			nState_DropCup := 6;
		ELSE
			tTimer_DropCup(IN := TRUE, PT := REAL_TO_TIME(timerCheckStuck)*1000);
			IF tTimer_DropCup.Q  THEN
				IF nLine = 1 THEN
					F_SetError(2,nLine := 1);
				ELSIF nLine = 2 THEN
					F_SetError(24,nLine := 2);
				END_IF
			END_IF
		END_IF
	6: //complete
		iCylinder_Dw.Extend();
		tTimer_DropCup(IN := TRUE, PT := REAL_TO_TIME(timerCheckCylinder_Dw)*1000);
		IF tTimer_DropCup.Q THEN
			IF nLine = 1 THEN
				F_SetError(5,nLine := 1);
			ELSIF nLine = 2 THEN
				F_SetError(27,nLine := 2);
			END_IF
		ELSIF iCylinder_Dw.bIsExtend THEN
			tTimer_DropCup(IN := FALSE);
			nState_DropCup := 7;
		END_IF
	7:
		iCylinder_Up.Retract();
		tTimer_DropCup(IN := TRUE, PT := REAL_TO_TIME(timerCheckCylinder_Up)*1000);
		IF tTimer_DropCup.Q THEN
			IF nLine = 1 THEN
				F_SetError(3,nLine := 1);
			ELSIF nLine = 2 THEN
				F_SetError(25,nLine := 2);
			END_IF
		ELSIF iCylinder_Up.bIsRetract THEN
			DropCup := TRUE;
			tTimer_DropCup(IN := FALSE);
			nState_DropCup := 0;
		END_IF
END_CASE
END_METHOD

METHOD Enable : BOOL
VAR_INPUT
END_VAR
CASE nState_Enable OF
	0:
		Enable := FALSE;
		tTimer_Enable1(IN := FALSE);
		tTimer_Enable2(IN := FALSE);
		nState_Enable := 1;
	1:
		iCylinder_Up.Retract();
		iCylinder_Dw.Extend();
		nState_Enable := 2;
	2:
		tTimer_Enable1(IN := TRUE, PT := REAL_TO_TIME(timerCheckCylinder_Up));
		tTimer_Enable2(IN := TRUE, PT := REAL_TO_TIME(timerCheckCylinder_Dw));
		IF tTimer_Enable1.Q AND NOT iCylinder_Up.bIsRetract THEN
			IF nLine = 1 THEN
				F_SetError(3,nLine := 1);
				nState_Enable := 99;//error
			ELSIF nLine = 2 THEN
				F_SetError(21,nLine := 2);
				nState_Enable := 99;//error
			END_IF
		ELSIF tTimer_Enable2.Q AND NOT iCylinder_Dw.bIsExtend THEN
			IF nLine = 1 THEN
				F_SetError(4,nLine := 1);
				nState_Enable := 99;//error
			ELSIF nLine = 2 THEN
				F_SetError(22,nLine := 2);
				nState_Enable := 99;//error
			END_IF
		ELSIF iCylinder_Up.bIsRetract AND iCylinder_Dw.bIsExtend THEN
			tTimer_Enable1(IN := FALSE);
			tTimer_Enable2(IN := FALSE);
			nState_Enable := 3;
		END_IF
	3:
		Enable := TRUE;
	99://Error
END_CASE
END_METHOD

METHOD HoldCup : BOOL
VAR_INPUT
END_VAR
iCylinder_Up.Extend();
END_METHOD

METHOD Init : BOOL
VAR_INPUT
END_VAR
nState_DropCup				:= 0;
nState_Enable				:= 0;
END_METHOD

PROPERTY isCupDrop : BOOL
GET
isCupDrop := bCupDrop;
END_GET
END_PROPERTY

PROPERTY isCupEmpty : BOOL
GET
isCupEmpty := bCupEmpty;
END_GET
END_PROPERTY

METHOD Manual : BOOL
VAR_INPUT
	bCylinder_up_extend 			: BOOL;
	bCylinder_up_retract 			: BOOL;
	bCylinder_dw_extend 			: BOOL;
	bCylinder_dw_retract 			: BOOL;
	bCylinder_suction_extend 		: BOOL;
	bCylinder_suction_retract 		: BOOL;
END_VAR

VAR
	re: INT;
END_VAR
IF bCylinder_up_extend THEN
	iCylinder_Up.Extend();
END_IF

IF bCylinder_up_retract THEN
	iCylinder_Up.Retract();
	tTimer_Up(IN := TRUE, PT := REAL_TO_TIME(timerCheckCylinder_Up)*1000);
		IF tTimer_Up.Q THEN
			IF nLine = 1 THEN
				F_SetError(3,nLine := 1);
			ELSIF nLine = 2 THEN
				F_SetError(25,nLine := 2);
			END_IF
		ELSIF iCylinder_Up.bIsRetract THEN
			tTimer_Up(IN := FALSE);
		END_IF
END_IF

IF bCylinder_dw_extend THEN
	iCylinder_Dw.Extend();
	tTimer_Dw(IN := TRUE, PT := REAL_TO_TIME(timerCheckCylinder_Dw)*1000);
		IF tTimer_Dw.Q THEN
			IF nLine = 1 THEN
				F_SetError(5,nLine := 1);
			ELSIF nLine = 2 THEN
				F_SetError(27,nLine := 2);
			END_IF
		ELSIF iCylinder_Dw.bIsExtend THEN
			tTimer_Dw(IN := FALSE);
		END_IF;
END_IF

IF bCylinder_dw_retract THEN
	iCylinder_Dw.Retract();
	tTimer_Dw(IN := TRUE, PT := REAL_TO_TIME(timerCheckCylinder_Dw)*1000);
		IF tTimer_Dw.Q THEN
			IF nLine = 1 THEN
				F_SetError(4,nLine := 1);
			ELSIF nLine = 2 THEN
				F_SetError(26,nLine := 2);
			END_IF
		ELSIF iCylinder_Dw.bIsRetract THEN
			tTimer_Dw(IN := FALSE);
		END_IF;
END_IF

IF bCylinder_suction_retract THEN
	iCylinder_Suction.Retract();
END_IF

IF bCylinder_suction_extend THEN
	iCylinder_Suction.Extend();
	tTimer_Suction(IN := TRUE, PT := REAL_TO_TIME(timerCylinder_Suction)*1000);
		IF tTimer_Suction.Q THEN
			IF nLine = 1 THEN
				F_SetError(60,nLine := 1);
			ELSIF nLine = 2 THEN
				F_SetError(61,nLine := 2);
			END_IF
		ELSIF iCylinder_Suction.bIsExtend THEN
			tTimer_Suction(IN := FALSE);
		END_IF
END_IF
END_METHOD

METHOD Reset : BOOL
VAR_INPUT
END_VAR
tTimer_DropCup(IN := FALSE);
tTimer_Enable1(IN := FALSE);
tTimer_Enable2(IN := FALSE);
iCylinder_Suction.Extend();
tTimer_Up(IN := FALSE);
tTimer_Dw(IN := FALSE);
tTimer_Suction(IN := FALSE);
CASE nState_Reset OF
	0:
		tTimer_Reset(IN := TRUE, PT := T#300MS);
		iCylinder_Dw.Extend();
		IF tTimer_Reset.Q OR iCylinder_Dw.bIsExtend THEN
			nState_Reset := 1;
		END_IF
	1:
		tTimer_Reset(IN := FALSE);
		iCylinder_Up.Retract();
		nState_Reset := 0;
END_CASE
END_METHOD

METHOD Stop : BOOL
VAR_INPUT
END_VAR
tTimer_Enable1(IN := FALSE);
tTimer_Enable2(IN := FALSE);
tTimer_DropCup(IN := FALSE);
tTimer_Up(IN := FALSE);
tTimer_Dw(IN := FALSE);
tTimer_Suction(IN := false);
iCylinder_Dw.Extend();
END_METHOD

END_FUNCTION_BLOCK

// ---- POUs/Components/Child Components/FB_Cylinder.TcPOU
FUNCTION_BLOCK FB_Cylinder IMPLEMENTS I_Cylinder
VAR_INPUT
	id	: INT;
END_VAR
VAR_OUTPUT
END_VAR
VAR
	bAtExtend 		AT %I*	: BOOL;
	bAtRetract 		AT %I*	: BOOL;
	bAtRetract_2	AT %I*	: BOOL;
	bMoveExtend 	AT %Q*	: BOOL;
	bMoveRetract 	AT %Q*	: BOOL;
END_VAR

PROPERTY bIsExtend : BOOL
GET
bIsExtend := bAtExtend;
END_GET
END_PROPERTY

PROPERTY bIsRetract : BOOL
GET
bIsRetract := bAtRetract;
END_GET
END_PROPERTY

METHOD Extend : BOOL
VAR_INPUT
END_VAR
bMoveExtend := TRUE;
bMoveRetract := FALSE;
END_METHOD

METHOD Retract : BOOL
VAR_INPUT
END_VAR
bMoveExtend := FALSE;
bMoveRetract := TRUE;
END_METHOD

END_FUNCTION_BLOCK

// ---- POUs/Components/Sim Components/FB_Cylinder_Sim.TcPOU
FUNCTION_BLOCK FB_Cylinder_Sim IMPLEMENTS I_Cylinder
VAR_INPUT
END_VAR
VAR_OUTPUT
END_VAR
VAR
	// original IO
	bAtExtend 		: BOOL;
	bAtRetract 		: BOOL;
	bMoveExtend 	: BOOL;
	bMoveRetract 	: BOOL;
	// internal vars for simulation
	fbTimer				: TON;
	tDelay				: TIME := T#1000MS;
	bStartAtRetractPos	: BOOL := TRUE; // TRUE if default pos is at retract pos
	nState				: INT := 0;
END_VAR

CASE nState OF
	0: // init start position sensor
	IF bStartAtRetractPos THEN
		bAtRetract := TRUE;
	ELSE
		bAtExtend := TRUE;
	END_IF
	nState := nState + 1;
	
	1: // check for move signal
	IF (bMoveExtend AND bAtRetract) THEN
		nState := 10;
	END_IF
	IF (bMoveRetract AND bAtExtend) THEN
		nState := 20;
	END_IF
	
	10: // move to extend pos
	bAtRetract := FALSE;
	fbTimer(IN:=TRUE, PT:=tDelay);
	IF fbTimer.Q THEN
		fbTimer(IN:=FALSE);
		bAtExtend := TRUE;
		nState := 1;
	END_IF
	
	20: // move to retract pos
	bAtExtend := FALSE;
	fbTimer(IN:=TRUE, PT:=tDelay);
	IF fbTimer.Q THEN
		fbTimer(IN:=FALSE);
		bAtRetract := TRUE;
		nState := 1;
	END_IF
	
END_CASE

PROPERTY bIsExtend : BOOL
GET
bIsExtend := bAtExtend;
END_GET
END_PROPERTY

PROPERTY bIsRetract : BOOL
GET
bIsRetract := bAtRetract;
END_GET
END_PROPERTY

METHOD Extend : BOOL
VAR_INPUT
END_VAR
bMoveExtend := TRUE;
bMoveRetract := FALSE;
END_METHOD

METHOD Retract : BOOL
VAR_INPUT
END_VAR
bMoveExtend := FALSE;
bMoveRetract := TRUE;
END_METHOD

END_FUNCTION_BLOCK

// ---- POUs/Functions/F_SetWarning.TcPOU
FUNCTION F_SetWarning : BOOL
VAR_INPUT
	nWrningID	: INT;
	nLine		: INT;
END_VAR
VAR
END_VAR

IF nLine = 1 THEN
	bWarning  := TRUE;
ELSIF nLine = 2 THEN
	bWarning2 := TRUE;
END_IF
nWarningID	:= nWrningID;

END_FUNCTION

// ---- POUs/Modules/FB_FoodWeightModule.TcPOU
FUNCTION_BLOCK FB_FoodWeightModule
VAR_INPUT
	nLine					: INT;
	UnitID					: BYTE;
	fFast_Speed				: REAL;
	fSlow_Speed_1			: REAL;
	fSlow_Speed_2			: REAL;
	fDerisedWeight_Food		: REAL;
	fChangeMode_Food_1		: REAL;
	fChangeMode_Food_2		: REAL;
	fMaxWeight_Food			: REAL;
	fPerStop_Food			: REAL;
	fTimer_Food				: REAL;
	fTimer_Alarm_Food		: REAL;
	fTimer_Check_Food		: REAL;
	fTimer_Error_Food		: REAL;
	fDelta_Food				: REAL;
	fTimer_Reverse			: REAL;
END_VAR
VAR_OUTPUT
	fProductLogF			: ARRAY [1..5] OF REAL;
	bStatus_Food			: BOOL;
	Time_start				: DT;
	Time_Stop				: DT;
	status					: STRING;
	fweight_iot				: REAL;
END_VAR
VAR
	// ===== CHILD COMPONENTS ============
	fbDriver			: FB_Inverter;
	fbLoadcell			: FB_Loadcell;
	// ===== SIM COMPONENTS ==============
	fbDriverSim			: FB_Inverter_Sim;
	fbLoadcellSim		: FB_LoadCell_Sim;
	// ===== INTERFACES ==================
	iDriver				: I_Inverter;
	iLoadcell			: I_LoadCell;
	// ====== VAR IO =====================
	bCupPresent 	AT %I*	: BOOL;
	bError_Driver   AT %I* 	: BOOL;
	//======= VAR METHOD =================
	nState				: INT;
	nStateErr			: INT;
	nStateWrn			: INT;
	fbTimer				: TON;
	fbTimer1			: TON;
	fbTimer_Alarm		: TON;
	fbTimer_Error		: TON;			
	fFastWeight			: REAL;
	fSlowWeight			: REAL;
	fSlowWeight1		: REAL;
	fChangemode_val		: REAL;
	fChangemode_val1	: REAL;
	fLowToleWeight		: REAL;
	fHighToleWeight		: REAL;
	fTareWeight			: REAL;
	bDone				: BOOL;
	p,k					: INT;
	//========= VAR HMI Worm Weight Auto ============
	fFlow_Food						: REAL;
	fWeight_Food					: REAL;
	fActDelta_Food					: REAL;	
	fSpeed_Food_Motor_Manual		: REAL;
	fTime							: REAL;
	Error							: BOOL;
	bStatus							: BOOL;
	timestart						: dt;
END_VAR

IF bSimMode THEN
	iDriver	:= fbDriverSim;
	fbDriverSim();
	iLoadcell	:= fbLoadcellSim;
	fbLoadcellSim();
ELSE
	iDriver	:= fbDriver;
	fbDriver(UnitID := UnitID, id := 2);
	iLoadcell	:= fbLoadcell;
	fbLoadcell(idDevice := nLine,Error => Error);
END_IF

IF iLoadcell.fActWeight > fMaxWeight_Food THEN
	IF nLine = 1 THEN
		F_SetError(56,nLine := 1);
	ELSIF nLine = 2 THEN
		F_SetError(58,nLine := 2);
	END_IF
END_IF

IF Error THEN
	IF nLine = 1 THEN
		F_SetError(69,nLine := 1);
	ELSIF nLine = 2 THEN
		F_SetError(71,nLine := 2);
	END_IF
END_IF

IF bIsError_Driver THEN
	iDriver.Stop();
	IF nLine = 1 THEN
		F_SetError(7,nLine := 1);
	ELSIF nLine = 2 THEN
		F_SetError(29,nLine := 2);
	END_IF
END_IF

METHOD Auto : BOOL
VAR_INPUT
END_VAR

VAR
END_VAR
GetLocalSystemTime(bEnable := 1);
fbTimer(PT := T#100S);
fbTimer_Alarm(PT := REAL_TO_TIME(fTimer_Alarm_Food)*1000);
CASE nState OF
	0:// Init Value
		Auto					:= FALSE;
		fbTimer(IN := FALSE);
		fbTimer1(IN := FALSE);
		fbTimer_Alarm(IN := FALSE);
		fbTimer_Error(IN := FALSE);
		bDone					:= FALSE;
		iDriver.fTargetSpeed 	:= fFast_Speed;
		nState 					:= 1;
	1:// Init Value
		fFastWeight				:= fFast_Speed;
		fSlowWeight				:= fSlow_Speed_1;
		fSlowWeight1			:= fSlow_Speed_2;
		fChangemode_val			:= fDerisedWeight_Food*fChangeMode_Food_1/100;
		fChangemode_val1		:= (fDerisedWeight_Food - fChangemode_val)*fChangeMode_Food_2/100 + fChangemode_val;
		fLowToleWeight			:= fDerisedWeight_Food*(1-(fDelta_Food/100));
		fHighToleWeight			:= fDerisedWeight_Food*(1+(fDelta_Food/100));
		bStatus_Food			:= FALSE;
		bStatus					:= FALSE;
		fTime					:= 0;
		nState					:= 2;
	2:// Cup detection
		iDriver.fTargetSpeed 	:= fFastWeight;
		iLoadcell.NetMode();
		IF NOT bIsCupPresent THEN
			fbTimer1(IN := TRUE, PT := REAL_TO_TIME(fTimer_Food)*1000);
			IF fbTimer1.Q THEN
				nState	:= 3;
			END_IF
		END_IF
	3:// Tare weight
		timestart := SYSTEMTIME_TO_DT(GetLocalSystemTime.systemTime);
		fbTimer1(IN := FALSE);
		fTareWeight 			:= iLoadcell.fActWeight;
		fWeight_Food			:= iLoadcell.fActWeight - fTareWeight;
		nState					:= 4;
	4:
		iDriver.Start();
		iDriver.fTargetSpeed	:= fSlowWeight;
		fbTimer_Alarm(IN := TRUE);
		fTime := TIME_TO_REAL(fbTimer.ET)/1000;
		fWeight_Food			:= iLoadcell.fActWeight - fTareWeight;
		fbTimer(IN := TRUE);
		fFlow_Food				:= fWeight_Food/((TIME_TO_REAL(fbTimer.ET)+0.00001)/1000);
		IF fWeight_Food >= fChangemode_val THEN
			nState 				:= 5;
		END_IF
	5:// Slow 1 Weight
		iDriver.Stop();
		nState					:= 55;
	55:
		iDriver.Start();
		iDriver.fTargetSpeed	:= fSlowWeight;
		fWeight_Food			:= iLoadcell.fActWeight	- fTareWeight;
		fbTimer(IN := TRUE);
		fTime := TIME_TO_REAL(fbTimer.ET)/1000;
		fFlow_Food				:= fWeight_Food/((TIME_TO_REAL(fbTimer.ET)+0.00001)/1000);
		IF fWeight_Food	>= fChangemode_val1 THEN
			nState				:= 6;
		END_IF
	6:// Slow 2 Weight
		iDriver.Stop();
		nState					:= 66;
	66:
		iDriver.fTargetSpeed	:= fSlowWeight1;
		iDriver.Start();
		fWeight_Food			:= iLoadcell.fActWeight	- fTareWeight;
		fbTimer(IN := TRUE);
		fTime := TIME_TO_REAL(fbTimer.ET)/1000;
		fFlow_Food				:= fWeight_Food/((TIME_TO_REAL(fbTimer.ET)+0.00001)/1000);
		IF fWeight_Food	>= fLowToleWeight*fPerStop_Food/100 THEN
			nState				:= 7;
		END_IF
	7:
		iDriver.Stop();
		nState					:= 71;
	71:
		iDriver.Reverse();
		fbTimer(IN := TRUE);
		fWeight_Food			:= iLoadcell.fActWeight	- fTareWeight;
		fbTimer1(IN := TRUE, PT := REAL_TO_TIME(fTimer_Reverse)*1000);
		fTime := TIME_TO_REAL(fbTimer.ET)/1000;
		IF fbTimer1.Q THEN
			nState 				:= 72;
		END_IF
	72:
		fbTimer1(IN := FALSE);
			nState				:= 73;
	73:// Wait Stable Weight
		iDriver.fTargetSpeed 	:= fFastWeight;
		iDriver.Stop();
		fTime := TIME_TO_REAL(fbTimer.ET)/1000;
		fbTimer(IN := TRUE);
		fWeight_Food			:= iLoadcell.fActWeight	- fTareWeight;
		fbTimer1(IN := TRUE, PT := REAL_TO_TIME(fTimer_Check_Food)*1000);
		IF fbTimer1.Q THEN
			nState				:= 8;
		END_IF
	8:// Check Done
		fbTimer1(IN := FALSE);
		fbTimer_Alarm(IN := TRUE);
		fWeight_Food			:= iLoadcell.fActWeight	- fTareWeight;
		IF fWeight_Food < fLowToleWeight THEN
			nState				:= 9;
		ELSIF fWeight_Food >= fLowToleWeight AND fWeight_Food <= fHighToleWeight THEN
			nState				:= 10;
		ELSIF fWeight_Food > fHighToleWeight THEN
			nState				:= 11;	
		END_IF
	9:// No Enough Weight
		fWeight_Food			:= iLoadcell.fActWeight - fTareWeight;
		iDriver.fTargetSpeed	:= fSlowWeight1;
		iDriver.Start();
		IF fWeight_Food	>= fLowToleWeight THEN
			nState				:= 7;
		END_IF
	10:// Enough Weight
		fActDelta_Food			:= (fWeight_food - fDerisedWeight_Food)/fDerisedWeight_Food*100;
		fWeight_Food			:= iLoadcell.fActWeight - fTareWeight;
		fweight_iot				:= iLoadcell.fActWeight - fTareWeight;
		Time_start				:= timestart;
		bStatus_Food			:= TRUE;
		status					:= 'Pass';
		fbTimer(IN := FALSE);
		fbTimer_Alarm(IN := FALSE);
		bDone					:= TRUE;
		p						:= p + 1;
		nState					:= 12;
	11:// Overweight
		fActDelta_Food			:= (fWeight_Food - fDerisedWeight_Food)/fDerisedWeight_Food*100;
		fWeight_Food			:= iLoadcell.fActWeight - fTareWeight;
		fweight_iot				:= iLoadcell.fActWeight - fTareWeight;
		Time_start				:= timestart;
		bStatus_Food			:= FALSE;
		status					:= 'Fail';
		fbTimer_Alarm(IN := FALSE);
		fbTimer(IN := FALSE);
		fbTimer_Error(IN := FALSE);
		bDone					:= TRUE;
		p						:= p + 1;
		IF nLine = 1 THEN
			//F_SetWarning(104);
			nState				:= 12;
		ELSIF nLine = 2 THEN
			//F_SetWarning(111);
			nState				:= 12;
		END_IF
	12:// Done
		Time_Stop				:= SYSTEMTIME_TO_DT(GetLocalSystemTime.systemTime);
		bStatus					:= TRUE;
		IF p > 5 THEN
			p := 5;
		END_IF
		IF bDone THEN
			IF p <> 1 THEN
				FOR k := p TO 2 BY -1 DO
					fProductLogF[k] := fProductLogF[k-1];
				END_FOR
			END_IF
			fProductLogF[1]	:= fWeight_Food;
			bDone 			:= FALSE;
		END_IF
		Auto					:= TRUE;
		nState					:= 13;
	13:
		nState					:= 0;
END_CASE

//Check Timer WormWeight
CASE nStateWrn OF 
	0:
		IF fbTimer_Alarm.Q THEN
			IF nLine = 1 THEN
				F_SetWarning(103,nLine := 1);
			ELSIF nLine = 2 THEN
				F_SetWarning(110,nLine := 2);
			END_IF
			nStateWrn := 1;
		END_IF
	1:
		IF NOT fbTimer_Alarm.Q THEN
			IF nLine = 1 THEN
				bWrn := FALSE;
			ELSIF nLine = 2 THEN
				bWrn2 := FALSE;
			END_IF
			bSirens := FALSE;
			nStateWrn := 0;
		END_IF
		fbTimer_Error(IN := TRUE, PT := REAL_TO_TIME(fTimer_Error_Food*1000));
		IF fbTimer_Error.Q THEN
			IF nLine = 1 THEN
				F_SetError(76,nLine := 1);
			ELSIF nLine = 2 THEN
				F_SetError(78,nLine := 2);
			END_IF
			fbTimer_Alarm(IN := FALSE);
			nState := 11;
			nStateWrn := 0;
		END_IF	
END_CASE

// Check Fault CupPresent

IF nState > 2 AND nState < 99 THEN
	IF bIsCupPresent THEN
		IF nLine = 1 THEN
			F_SetError(45,nLine := 1);
			nState := 0;
		ELSIF nLine = 2 THEN
			F_SetError(46,nLine := 2);
			nState := 0;
		END_IF
	END_IF
END_IF

// Write ProductLog
END_METHOD

PROPERTY bIsCupPresent : BOOL
GET
bIsCupPresent := bCupPresent;
END_GET
END_PROPERTY

PROPERTY bIsError_Driver : BOOL
GET
bIsError_Driver	:= bError_Driver;
END_GET
END_PROPERTY

METHOD Enable : BOOL
VAR_INPUT
END_VAR
iLoadcell.NetMode();
END_METHOD

METHOD Init : BOOL
VAR_INPUT
END_VAR
nState := 0;
END_METHOD

METHOD Manual : BOOL
VAR_INPUT
	bUp_Food_Motor					: BOOL;
	bDown_Food_Motor				: BOOL;
	bZero_Loadcell_Food				: BOOL;
	bMotor_Food						: BOOL;	
	bMotor_Food_Reverse				: BOOL;
END_VAR
IF bUp_Food_Motor THEN
	fSpeed_Food_Motor_Manual	:= fSpeed_Food_Motor_Manual + 10;
END_IF

IF bDown_Food_Motor THEN
	fSpeed_Food_Motor_Manual	:= fSpeed_Food_Motor_Manual - 10;
END_IF

IF bMotor_Food THEN
	iDriver.Start();
ELSIF bMotor_Food_Reverse THEN
	iDriver.Reverse();
ELSIF NOT bMotor_Food AND NOT bMotor_Food_Reverse THEN
	iDriver.Stop();
END_IF

iDriver.fTargetSpeed	:= fSpeed_Food_Motor_Manual;

IF bZero_Loadcell_Food THEN
	iLoadcell.Set_Zero();
ELSE
	iLoadcell.NetMode();
END_IF

fWeight_Food := iLoadcell.fActWeight;
END_METHOD

METHOD Reset : BOOL
VAR_INPUT
END_VAR
iDriver.Reset();
fbTimer(IN := FALSE);			
fbTimer1(IN	:= FALSE);
fbTimer_Alarm(IN := FALSE);
fbTimer_Error(IN := FALSE);
END_METHOD

METHOD SetZero : BOOL
VAR_INPUT
END_VAR
iLoadcell.Set_Zero();
END_METHOD

METHOD Stop : BOOL
VAR_INPUT
END_VAR
iDriver.Stop();
fbTimer(IN := FALSE);			
fbTimer1(IN	:= FALSE);
fbTimer_Alarm(IN := FALSE);
fbTimer_Error(IN := FALSE);
END_METHOD

END_FUNCTION_BLOCK

// ---- POUs/Components/Child Components/FB_Loadcell.TcPOU
FUNCTION_BLOCK FB_Loadcell IMPLEMENTS I_LoadCell
VAR_INPUT
	idDevice					: INT;// 1: mettler		,2: Laumas
END_VAR
VAR_OUTPUT
	Error						: BOOL;
END_VAR
VAR
	ondinh						: BOOL;
	fbInterface					: FB_Interface_EtherCat;
	nErrID						: INT;	
END_VAR

fbInterface(idDevice := idDevice,Error => Error);

PROPERTY fActWeight : REAL
GET
fActWeight := fbInterface.fActWeight;
END_GET
END_PROPERTY

METHOD NetMode : BOOL
VAR_INPUT
END_VAR
fbInterface.NetMode();
END_METHOD

METHOD Set_Zero : BOOL
VAR_INPUT
END_VAR
fbInterface.Set_Zero();
END_METHOD

PROPERTY Status : REAL;
GET
Status := fbInterface.Status;
END_GET
END_PROPERTY

END_FUNCTION_BLOCK

// ---- POUs/Components/Child Components/FB_Interface_EtherCat.TcPOU
FUNCTION_BLOCK FB_Interface_EtherCat
VAR_INPUT
    idDevice                : INT; // 1 : mettler    , 2: Laumas
END_VAR
VAR_OUTPUT
	Error					: BOOL;
END_VAR
VAR
    IND360_tareStableCMD    :    BOOL;
    IND360_tareImmediateCMD    :    BOOL;
    IND360_zeroStableCMD    :    BOOL;
    IND360_zeroImmediateCMD    :    BOOL;
    IND360_clearCMD            :    BOOL;
    IND360_preTareCMD        :    BOOL;
    IND360_preTareCMDVAL    :    REAL;
    IND360_reportedWeight    :    REAL;
    IND360_stableWeight        :    REAL;
    IND360_heartBeat        :    BOOL;
    IND360_DataOK            :    BOOL;
    IND360_Smart5lvl5        :    BOOL;
    IND360_Smart5lvl4        :    BOOL;
    IND360_Smart5lvl3        :    BOOL;
    IND360_Smart5lvl2        :    BOOL;
    IND360_centerofZero        :    BOOL;
    IND360_motion            :    BOOL;
    IND360_netMode            :    BOOL;
    IND360_cmdDone            :    BOOL;
    IND360_cmdPending        :    BOOL;
    IND360_cmdFailed        :    BOOL;
    IND360_weightCMD        :    UINT        := 3;
    //Variables and Function Block for SAI Device Heartbeat check
    IND360_Alive            :    BOOL;
    IND360_heartBeat_        :    BOOL;
    //EtherCAT device's CoE identification:
    IND360_NetId            :     T_AmsNetId     := '192.168.0.106.3.1'; // Have to be entered
    IND360_SlaveAddr         :     UINT         := 1001;     // Have to be entered        
    //Variables and Function Block for APW Internal Adjustment Procedure
    IntAdjust_Done            :    BOOL;
    IntAdjust_Error            :    BOOL;
    IntAdjust_Process        :    BOOL;
    IntAdjust_Cancelled        :    BOOL;
    IntAdjust_Start            :    BOOL;
    IntAdjust_Cancel        :    BOOL;
    //Variables and Function Block for APW External Adjustment Procedure    
    ExtAdjust_Done            :    BOOL;
    ExtAdjust_Error            :    BOOL;
    ExtAdjust_Process        :    BOOL;
    ExtAdjust_Cancelled        :    BOOL;
    ExtAdjust_Start            :    BOOL;
    ExtAdjust_Cancel        :    BOOL;
    ExtAdjust_Load            :    BOOL;
    ExtAdjust_Unload        :    BOOL;
    ExtAdjust_currWeight    :    REAL;
    ExtAdjust_extWeight        :    REAL;
    //IO
    //Var of FB SAI
    IND_M_WR_Float         AT %Q* : REAL; //write float to devices     
    IND_M_WR_Channel     AT %Q* : WORD; //select device to write    
    IND_M_WR_Command     AT %Q* : WORD; //command to device    
    IND_SB_RSV1             AT %Q* : WORD;
    IND_SB_RSV2             AT %Q* : WORD;
    IND_SB_RSV3             AT %Q* : WORD;
    IND_SB_CMD             AT %Q* : WORD;

 

 

    IND_M_RD_Float         AT %I* : REAL; //read float from devices
    IND_M_RD_Status         AT %I* : WORD; //read status of device    
    IND_M_RD_Response     AT %I* : INT;
    IND_SB_STT1             AT %I* : WORD;
    IND_SB_STT2             AT %I* : WORD;
    IND_SB_STT3             AT %I* : WORD;
    IND_SB_RSP             AT %I* : WORD;    

 

    //var Ext
    fbAdjust_CoESdoWrite_Ext    :     FB_EcCoESdoWrite;
    fbStatus_CoESdoRead_Ext        :    FB_EcCoESdoRead;
    fbWeight_CoESdoRead_Ext        :    FB_EcCoESdoRead;
    fbWeight_CoESdoWrite_Ext    :    FB_EcCoESdoWrite;
    fbCancel_CoESdoWrite_Ext    :     FB_EcCoESdoWrite;
    nState_Ext                :    SINT        :=    0;
    fbStart_RTrig_Ext        :    R_TRIG;
    fbCancel_RTrig_Ext        :    R_TRIG;
    wValue_Ext                :    BYTE        :=    1;
    wValue0_Ext                :    BYTE        :=    0;
    iStatus_Ext                :    INT;
    bRead_Ext                :    BOOL;
    bRead2_Ext                :    BOOL;
    bWrite_Ext                :    BOOL;
    fbtimer_Ext                :    TON;
    currentWeight0_Ext        :    REAL;
    //var int
    fbAdjust_CoESdoWrite_Int    :     FB_EcCoESdoWrite;
    fbStatus_CoESdoRead_Int        :    FB_EcCoESdoRead;
    fbCancel_CoESdoWrite_Int    :     FB_EcCoESdoWrite;
    nState_Int                :    SINT        :=    0;
    fbStart_RTrig_Int        :    R_TRIG;
    fbCancel_RTrig_Int        :    R_TRIG;
    wValue_Int                :    BYTE        :=    1;
    rValue_Int                :    INT;
    bRead_Int                :    BOOL;
    bWrite_Int                :    BOOL;
    fbtimer_Int                :    TON;
    //var check
    heartBeatRTrig_Check        :    R_TRIG;
    heartBeatFTrig_Check        :    F_TRIG;
    timerReset_Check            :    BOOL;
    timer2S_Check                :    TON;
    //var weight
    writeTrigger_W            :    BOOL;
    restoreTrigger_W        :    BOOL;
    cmd_W                    :    UINT;
    fbRTrig_TareStable_W    :     R_TRIG;
    fbRTrig_TareImm_W        :    R_TRIG;
    fbRTrig_ZeroStable_W    :    R_TRIG;
    fbRTrig_ZeroImm_W        :    R_TRIG;
    fbRTrig_PreTare_W        :    R_TRIG;
    fbRTrig_Clear_W            :    R_TRIG;
    sequence0_W                :    BOOL;
    sequence1_W                :    BOOL;

    //=======var laumas=======
    CMDLaumas        AT %Q*    :     BYTE;
    WeightLaumas1    AT %I*    :     BYTE;//address 0x0004
    WeightLaumas2    AT %I*    :     BYTE;//address 0x0005
    WeightLaumas3    AT %I*    :     BYTE;//address 0x0006
    WeightLaumas4    AT %I*    :     BYTE;//address 0x0007
    StatusLaumas1    AT %I*    :     BYTE;//address 0x0012
    StatusLaumas2    AT %I*    :     BYTE;//address 0x0013

    uWeightLaumas            :     U_4Bytes2Real;
    uStatusLaumas            :     U_4Bytes2Real;
END_VAR

SAI_APW_ExtAdjust(
	deviceNetId:= IND360_NetId, 
	deviceSlaveAddr:= IND360_SlaveAddr, 
	currentWeight=> ExtAdjust_currWeight, 
	Load_Weight=> ExtAdjust_Load, 
	Unload_Weight=> ExtAdjust_Unload, 
	Process=> ExtAdjust_Process, 
	Done=> ExtAdjust_Done, 
	Error=> ExtAdjust_Error, 
	Cancelled=> ExtAdjust_Cancelled, 
	externalWeight:= ExtAdjust_extWeight, 
	Start:= ExtAdjust_Start, 
	Cancel:= ExtAdjust_Cancel);
	

SAI_APW_IntAdjust(
	deviceNetId:= IND360_NetId, 
	deviceSlaveAddr:= IND360_SlaveAddr, 
	Process=> IntAdjust_Process, 
	Done=> IntAdjust_Done, 
	Error=> IntAdjust_Error, 
	Cancelled=> IntAdjust_Cancelled, 
	Start:= IntAdjust_Start, 
	Cancel:= IntAdjust_Cancel);
	
SAI_Cyclic_CheckAlive(
	MB_DeviceStatus:= IND_M_RD_Status, 
	Alive=> IND360_Alive, 
	HeartBeat=> IND360_heartBeat_);
	
SAI_Cyclic_WeightProc(
	weightCmd:= IND360_weightCMD, 
	MB_DeviceStatus:= IND_M_RD_Status, 
	realtimeWeight=> IND360_reportedWeight, 
	stableWeight=> IND360_stableWeight, 
	heartBeat=> IND360_heartBeat, 
	DataOK=> IND360_DataOK, 
	Smart5_red=> IND360_Smart5lvl5, 
	Smart5_orange=> IND360_Smart5lvl4, 
	Smart5_yellow=> IND360_Smart5lvl3, 
	Smart5_blue=> IND360_Smart5lvl2, 
	centerofZero=> IND360_centerofZero, 
	motion=> IND360_motion, 
	netMode=> IND360_netMode, 
	cmdDone=> IND360_cmdDone, 
	cmdPending=> IND360_cmdPending, 
	cmdFailed=> IND360_cmdFailed, 
	TareStable_cmd:= IND360_tareStableCMD, 
	TareImmediate_cmd:= IND360_tareImmediateCMD, 
	ZeroStable_cmd:= IND360_zeroStableCMD, 
	ZeroImmediate_cmd:= IND360_zeroImmediateCMD, 
	PreTare_cmd:= IND360_preTareCMD, 
	PreTare_value:= IND360_preTareCMDVAL, 
	Clear_cmd:= IND360_clearCMD, 
	MB_MeasuredValue:= IND_M_RD_Float, 
	MB_Response:= IND_M_RD_Response, 
	MB_CmdValue:= IND_M_WR_Float, 
	MB_Command:= IND_M_WR_Command);
	
//Error Mettler
IF idDevice = 1 THEN
	IF IND360_Alive = 0 THEN
		Error := TRUE;
	ELSIF IND_SB_STT1.0 = 1 THEN
		Error := TRUE;
	ELSIF IND_SB_STT1.1 = 1 THEN
		Error := TRUE;
	ELSIF IND_SB_STT1.2 = 1 THEN
		Error := TRUE;
	ELSIF IND_SB_STT1.3 = 1 THEN
		Error := TRUE;
	ELSIF IND_SB_STT1.4 = 1 THEN
		Error := TRUE;
	ELSIF IND_SB_STT1.5 = 1 THEN
		Error := TRUE;
	ELSIF IND_SB_STT1.7 = 1 THEN
		Error := TRUE;
	ELSIF IND_SB_STT1.8 = 1 THEN
		Error := TRUE;
	ELSIF IND_SB_STT1.13 = 1 THEN
		Error := TRUE;
	ELSE
		Error := FALSE;
	END_IF
ELSIF idDevice = 2 THEN
	IF StatusLaumas1.0 = 1 THEN
		Error := TRUE;
	ELSIF StatusLaumas2.7 = 1 THEN
		Error := TRUE;
	ELSE
		Error := FALSE;
	END_IF
END_IF



// link Laumas
uWeightLaumas.st4bytes.Byte1 := WeightLaumas1;
uWeightLaumas.st4bytes.Byte2 := WeightLaumas2;
uWeightLaumas.st4bytes.Byte3 := WeightLaumas3;
uWeightLaumas.st4bytes.Byte4 := WeightLaumas4;

 

uStatusLaumas.st4bytes.Byte1 := StatusLaumas1;
uStatusLaumas.st4bytes.Byte2 := StatusLaumas2;

PROPERTY fActWeight : REAL
GET
IF idDevice = 1 THEN
    fActWeight := IND_M_RD_Float;
ELSIF idDevice = 2 THEN
	IF StatusLaumas2.0 = 1 THEN
		 fActWeight := -DINT_TO_REAL(uWeightLaumas.fReal)/100;
	ELSE
		fActWeight := DINT_TO_REAL(uWeightLaumas.fReal)/100;
	END_IF
END_IF
END_GET
END_PROPERTY

METHOD NetMode : BOOL
VAR_INPUT
END_VAR
IF idDevice = 1 THEN
    IND_M_WR_Command := 3;
ELSIF idDevice = 2 THEN
    CMDLaumas := 9;
END_IF
END_METHOD

METHOD SAI_APW_ExtAdjust
VAR_INPUT
   	deviceNetId         : 	T_AmsNetId 	:= '192.168.0.106.3.1'; // Have to be entered
  	deviceSlaveAddr     : 	UINT 		:= 1001;     // Have to be entered		
END_VAR
VAR_OUTPUT
	currentWeight		:	REAL;		//current adjustment weight to be loaded onto the scale
	Load_Weight			:	BOOL;		//flag to load the adjustment weight according to currentWeight
	Unload_Weight		:	BOOL;		//flag to unload the weight from the scale
	Process				:	BOOL;
	Done				: 	BOOL;
	Error				:	BOOL;
	Cancelled			:	BOOL;
END_VAR
VAR_IN_OUT
	externalWeight		:	REAL;
	Start				: 	BOOL;	
	Cancel				:	BOOL;
END_VAR
fbStart_RTrig_Ext(CLK:= Start, Q=> );
IF fbStart_RTrig_Ext.Q THEN
	fbAdjust_CoESdoWrite_Ext(bExecute:= FALSE);
	fbWeight_CoESdoWrite_Ext(bExecute := FALSE);
	fbCancel_CoESdoWrite_Ext(bExecute := FALSE);
	Process			:=	FALSE;
	Error			:=	FALSE;
	Done			:=	FALSE;
	Cancelled		:=	FALSE;
	nState_Ext			:=	1;
END_IF

// Read the adjustment status CoE #4007 INT continuously
IF nState_Ext >= 4 THEN
	IF NOT fbStatus_CoESdoRead_Ext.bBusy THEN
		bRead_Ext	:= TRUE;
	ELSE
		bRead_Ext	:= FALSE;
	END_IF
	// Read CoE Index #4007 size of 2 bytes: 2047-inProcee; 0-Done
	fbStatus_CoESdoRead_Ext(
		sNetId		:= deviceNetId, 
		nSlaveAddr	:= deviceSlaveAddr, 
		nSubIndex	:= 0, 
		nIndex		:= 16#4007,
		pDstBuf		:= ADR(iStatus_Ext), 
		cbBufLen	:= SIZEOF(iStatus_Ext), 
		bExecute	:= bRead_Ext, 
		tTimeout	:= T#2S
		);	
		
	IF NOT fbWeight_CoESdoRead_Ext.bBusy THEN
		bRead2_Ext	:= TRUE;
	ELSE
		bRead2_Ext	:= FALSE;
	END_IF
	// Read the required external weight CoE #4011 4-byte REAL continuously
	fbWeight_CoESdoRead_Ext(
		sNetId		:= deviceNetId, 
		nSlaveAddr	:= deviceSlaveAddr, 
		nSubIndex	:= 0, 
		nIndex		:= 16#4011,
		pDstBuf		:= ADR(currentWeight0_Ext), 
		cbBufLen	:= SIZEOF(currentWeight0_Ext), 
		bExecute	:= bRead2_Ext, 
		tTimeout	:= T#2S
		);
END_IF

// Cancel adjustment procedure:
fbCancel_RTrig_Ext(CLK:=Cancel, Q=> );
wValue_Ext	:= 1;
fbCancel_CoESdoWrite_Ext(
	sNetId		:= deviceNetId, 
	nSlaveAddr	:= deviceSlaveAddr, 
	nSubIndex	:= 0, 
	nIndex		:= 16#4004, 
	pSrcBuf		:= ADR(wValue_Ext), 
	cbBufLen	:= SIZEOF(wValue_Ext), 
	bExecute	:= bWrite_Ext, 
	tTimeout	:= T#1S, 
	bBusy=> , 
	bError=> , 
	nErrId=> );

IF fbCancel_RTrig_Ext.Q THEN
	bWrite_Ext	:= TRUE;
END_IF

IF fbCancel_CoESdoWrite_Ext.bExecute = TRUE AND NOT fbCancel_CoESdoWrite_Ext.bBusy THEN
	iStatus_Ext			:=	0;
	Start			:=	FALSE;
	bWrite_Ext			:= 	FALSE;
	Process			:=	FALSE;
	Error			:=	FALSE;
	Cancelled		:=	TRUE;
	Done			:=	FALSE;
	Cancel			:=	FALSE;
	Load_Weight		:=	FALSE;
	Unload_Weight	:=	FALSE;
	currentWeight	:=	0.0;
	nState_Ext			:=	0;
END_IF

CASE nState_Ext OF
	1:
	IF externalWeight > 0.0 THEN
		nState_Ext	:= 2;
	ELSE 
		nState_Ext	:= 99;
	END_IF
	
	2:
	// Turn off the adjustment step control #401F 2-Byte CoE
	wValue0_Ext	:= 0;
	fbAdjust_CoESdoWrite_Ext(
	sNetId		:= deviceNetId,
	nSlaveAddr	:= deviceSlaveAddr,
	nSubIndex	:= 16#00,
	nIndex		:= 16#401F,
	pSrcBuf		:= ADR(wValue0_Ext),
	cbBufLen	:= SIZEOF(wValue0_Ext),
	bExecute	:= TRUE,
	tTimeout	:= T#1S
	);
	IF fbAdjust_CoESdoWrite_Ext.bError THEN
		nState_Ext	:= 99;
	ELSE
		IF NOT fbAdjust_CoESdoWrite_Ext.bBusy THEN
			iStatus_Ext			:=	0;
			currentWeight0_Ext	:=	0.0;
			nState_Ext			:= 3;
		END_IF
	END_IF
	
	3:	
	fbAdjust_CoESdoWrite_Ext(bExecute := FALSE);
	//write external weight into Index #4009, 4 bytes of REAL
	fbWeight_CoESdoWrite_Ext(
	sNetId		:= deviceNetId,
	nSlaveAddr	:= deviceSlaveAddr,
	nSubIndex	:= 16#00,
	nIndex		:= 16#4009,
	pSrcBuf		:= ADR(externalWeight),
	cbBufLen	:= SIZEOF(externalWeight),
	bExecute	:= TRUE,
	tTimeout	:= T#1S
	);
	IF fbWeight_CoESdoWrite_Ext.bError THEN
		nState_Ext	:= 99;
	ELSE
		IF NOT fbWeight_CoESdoWrite_Ext.bBusy THEN
			nState_Ext	:= 4;
		END_IF
	END_IF
	
	4:	//trigger the external adjustment process Index #4002, 1 byte data: [0000 0001]
	fbWeight_CoESdoWrite_Ext(bExecute := FALSE);
	fbtimer_Ext(IN:=FALSE,PT:=T#1000MS,Q=>,ET=>);
	fbAdjust_CoESdoWrite_Ext(
	sNetId		:= deviceNetId,
	nSlaveAddr	:= deviceSlaveAddr,
	nSubIndex	:= 16#00,
	nIndex		:= 16#4002,
	pSrcBuf		:= ADR(wValue_Ext),
	cbBufLen	:= SIZEOF(wValue_Ext),
	bExecute	:= TRUE,
	tTimeout	:= T#1S
	);
	IF fbAdjust_CoESdoWrite_Ext.bError THEN
		nState_Ext	:= 99;
	ELSE
		IF NOT fbAdjust_CoESdoWrite_Ext.bBusy THEN
			nState_Ext	:= 5;
		END_IF
	END_IF
	
	5:	
	fbtimer_Ext(IN:=TRUE,PT:=T#2000MS,Q=>,ET=>);
	fbAdjust_CoESdoWrite_Ext(bExecute:= FALSE);
	IF fbtimer_Ext.Q THEN
		IF iStatus_Ext	= 2046 THEN
			IF currentWeight0_Ext = 0.0 THEN
				nState_Ext := 5;
			ELSIF currentWeight0_Ext = externalWeight THEN
				nState_Ext := 6; 
			END_IF
		ELSIF iStatus_Ext < 0 THEN
			nState_Ext	:= 99;
		END_IF
	END_IF
	6:	
	fbtimer_Ext(IN:=FALSE,PT:=T#1000MS,Q=>,ET=>);
	IF iStatus_Ext	= 2046 THEN
		IF currentWeight0_Ext = 0.0 THEN
			nState_Ext := 7;
		ELSIF currentWeight0_Ext = externalWeight THEN
			nState_Ext := 6; 
		END_IF
	ELSIF iStatus_Ext < 0 THEN
		nState_Ext	:= 99;
	END_IF
	7:	
	IF currentWeight0_Ext	= 0.0 THEN
		IF iStatus_Ext = 0 THEN
			nState_Ext := 8;
		ELSIF iStatus_Ext = 2046 THEN
			nState_Ext := 7;
		ELSIF iStatus_Ext < 0 THEN
			nState_Ext	:= 99; 
		END_IF
	END_IF	
	
	8:
	fbtimer_Ext(IN:=TRUE,PT:=T#1000MS,Q=>,ET=>);
	IF fbtimer_Ext.Q THEN
		Error		:= FALSE;
		Process		:= FALSE;
		Done		:= TRUE;
		Start		:= FALSE;
		Cancelled	:= FALSE;	
		Load_Weight	:=	FALSE;
		Unload_Weight	:=	FALSE;
		nState_Ext		:= 0;
	END_IF
	
	99:	//error case
	currentWeight0_Ext	:= 0.0;
	Error		:= TRUE;
	Process		:= FALSE;
	Done		:= FALSE;
	Start		:= FALSE;
	Cancelled	:= FALSE;
	Load_Weight	:=	FALSE;
	Unload_Weight	:=	FALSE;
	nState_Ext 		:= 0;     // Error case	
END_CASE

// control the Load_Weight, Unload_Weight and Process flags
IF nState_Ext >= 4 AND nState_Ext < 8 AND NOT Cancel THEN
	IF iStatus_Ext = 2047 THEN
		Process		:=	TRUE;
	ELSE
		Process		:=	FALSE;
	END_IF
	
	IF iStatus_Ext = 2046 AND currentWeight0_Ext = externalWeight THEN
		Load_Weight		:=	TRUE;
	ELSE
		Load_Weight		:=	FALSE;
	END_IF

	IF currentWeight0_Ext = 0.0 THEN
		Unload_Weight		:=	TRUE;
	ELSE
		Unload_Weight		:=	FALSE;
	END_IF	
END_IF

// assign the VAR currentWeight0 to VAR_OUT currentWeight
currentWeight := currentWeight0_Ext;
END_METHOD

METHOD SAI_APW_IntAdjust : BOOL
VAR_INPUT
   	deviceNetId         : 	T_AmsNetId 	:= '192.168.0.106.3.1'; // Have to be entered
  	deviceSlaveAddr     : 	UINT 		:= 1001;     // Have to be entered		
END_VAR
VAR_OUTPUT
	Process				:	BOOL;
	Done				: 	BOOL;
	Error				:	BOOL;
	Cancelled			:	BOOL;
END_VAR
VAR_IN_OUT
	Start				: 	BOOL;	
	Cancel				:	BOOL;
END_VAR
fbStart_RTrig_Int(CLK:= Start, Q=> );
IF fbStart_RTrig_Int.Q THEN
	fbAdjust_CoESdoWrite_Int(bExecute:= FALSE);
	Process			:=	FALSE;
	Error			:=	FALSE;
	Done			:=	FALSE;
	Cancelled		:=	FALSE;
	nState_Int			:=	1;
END_IF

// Cancel adjustment procedure:
fbCancel_RTrig_Int(CLK:=Cancel, Q=> );
wValue_Int	:= 1;
fbCancel_CoESdoWrite_Int(
	sNetId		:= deviceNetId, 
	nSlaveAddr	:= deviceSlaveAddr, 
	nSubIndex	:= 0, 
	nIndex		:= 16#4004, 
	pSrcBuf		:= ADR(wValue_Int), 
	cbBufLen	:= SIZEOF(wValue_Int), 
	bExecute	:= bWrite_Int, 
	tTimeout	:= T#1S, 
	bBusy=> , 
	bError=> , 
	nErrId=> );

IF fbCancel_RTrig_Int.Q THEN
	bWrite_Int	:= TRUE;
END_IF

IF fbCancel_CoESdoWrite_Int.bExecute = TRUE AND NOT fbCancel_CoESdoWrite_Int.bBusy THEN
	rValue_Int			:=	0;
	Start			:=	FALSE;
	bWrite_Int			:= 	FALSE;
	Process			:=	FALSE;
	Error			:=	FALSE;
	Cancelled		:=	TRUE;
	Done			:=	FALSE;
	Cancel			:=	FALSE;
	nState_Int			:=	0;
END_IF

CASE nState_Int OF
	1:
		wValue_Int	:= 1;
		// Write byte data "16#01" into CoE Index #4001
	   	fbAdjust_CoESdoWrite_Int(
	   	sNetId		:= deviceNetId,
	   	nSlaveAddr	:= deviceSlaveAddr,
	   	nSubIndex	:= 16#00,
	   	nIndex		:= 16#4001,
	   	pSrcBuf		:= ADR(wValue_Int),
	   	cbBufLen	:= SIZEOF(wValue_Int),
	   	bExecute	:= TRUE,
	   	tTimeout	:= T#1S
	   	);
		nState_Int		:=	2;
	2:
	   	fbAdjust_CoESdoWrite_Int();       // Execute CoE write until done
   		IF fbAdjust_CoESdoWrite_Int.bError THEN
			Error	:= TRUE;
			Process	:= FALSE;
			Done	:= FALSE;
			Start	:= FALSE;
      		nState_Int 	:= 0;     // Error case
   		ELSE
			IF NOT fbAdjust_CoESdoWrite_Int.bBusy THEN
				nState_Int := 3;    
      		END_IF
   		END_IF
	3:
		IF NOT fbStatus_CoESdoRead_Int.bBusy THEN
			bRead_Int	:= TRUE;
		ELSE
			bRead_Int 	:= FALSE;
		END_IF
		// Read CoE Index #4007 size of 2 bytes: 2047-inProcee; 0-Done
		fbStatus_CoESdoRead_Int(
		sNetId		:= deviceNetId, 
		nSlaveAddr	:= deviceSlaveAddr, 
		nSubIndex	:= 0, 
		nIndex		:= 16#4007,
		pDstBuf		:= ADR(rValue_Int), 
		cbBufLen	:= SIZEOF(rValue_Int), 
		bExecute	:= bRead_Int, 
		tTimeout	:= T#1S
		);			

		fbtimer_Int(IN:= TRUE, PT:=T#1000MS, Q=> , ET=>);
		IF fbtimer_Int.Q AND NOT fbStatus_CoESdoRead_Int.bBusy THEN
			IF rValue_Int = 2047 THEN
				Error		:= FALSE;
				Process		:= TRUE;
				Done		:= FALSE;	
				Cancelled	:= FALSE;	
				nState_Int		:= 3;	
			ELSIF rValue_Int <0 THEN
				Error		:= TRUE;
				Process		:= FALSE;
				Done		:= FALSE;
				Start		:= FALSE;
				Cancelled	:= FALSE;
				nState_Int 		:= 0;     // Error case			
			ELSIF rValue_Int = 0 THEN
				Error		:= FALSE;
				Process		:= FALSE;
				Done		:= TRUE;
				Start		:= FALSE;
				Cancelled	:= FALSE;	
				nState_Int		:= 0;					
			END_IF
		END_IF
END_CASE
END_METHOD

METHOD SAI_Cyclic_CheckAlive : BOOL
VAR_INPUT
	MB_DeviceStatus		:	WORD;
END_VAR
VAR_OUTPUT
	Alive				:	BOOL;
	HeartBeat			:	BOOL;
END_VAR
HeartBeat	:=		MB_DeviceStatus.2;
heartBeatRTrig_Check(CLK := HeartBeat, Q => );
heartBeatFTrig_Check(CLK := HeartBeat, Q => );
timer2S_Check(IN:= NOT timerReset_Check, PT := T#2S, Q => , ET => );

IF heartBeatRTrig_Check.Q OR heartBeatFTrig_Check.Q THEN
	timerReset_Check	:= TRUE;
ELSE
	timerReset_Check	:= FALSE;
END_IF

IF timer2S_Check.Q THEN
	Alive	:= FALSE;
ELSE
	Alive	:= TRUE;
END_IF
END_METHOD

METHOD SAI_Cyclic_WeightProc : BOOL
VAR_INPUT
	weightCmd			:	UINT	:= 3;
	MB_DeviceStatus		:	WORD;	
END_VAR

VAR_OUTPUT
	realtimeWeight		:	REAL;
	stableWeight		:	REAL;
	heartBeat			:	BOOL;
	DataOK				:	BOOL;
	Smart5_red			:	BOOL;
	Smart5_orange		:	BOOL;
	Smart5_yellow		:	BOOL;
	Smart5_blue			:	BOOL;
	centerofZero		:	BOOL;
	motion				:	BOOL;
	netMode				:	BOOL;
	cmdDone				:	BOOL;
	cmdPending			:	BOOL;
	cmdFailed			:	BOOL;
END_VAR

VAR_IN_OUT
	TareStable_cmd		:	BOOL;
	TareImmediate_cmd	:	BOOL;
	ZeroStable_cmd		:	BOOL;
	ZeroImmediate_cmd	:	BOOL;
	PreTare_cmd			:	BOOL;
	PreTare_value		:	REAL;
	Clear_cmd			:	BOOL;
	MB_MeasuredValue	:	REAL;
	MB_Response			:	INT;
	MB_CmdValue			:	REAL;
	MB_Command			:	WORD;	
END_VAR
//List of most commonly used cyclic scale commands:
fbRTrig_TareStable_W(CLK:= TareStable_cmd, Q=> );
fbRTrig_TareImm_W(CLK:= TareImmediate_cmd, Q=> );
fbRTrig_ZeroStable_W(CLK:= ZeroStable_cmd, Q=> );
fbRTrig_ZeroImm_W(CLK:= ZeroImmediate_cmd, Q=> );
fbRTrig_PreTare_W(CLK:= PreTare_cmd, Q=> );
fbRTrig_Clear_W(CLK:= Clear_cmd, Q=> );

IF fbRTrig_TareStable_W.Q THEN
	cmd_W 			:= 400;
	writeTrigger_W	:= TRUE;
END_IF

IF fbRTrig_TareImm_W.Q THEN
	cmd_W 			:= 403;
	writeTrigger_W	:= TRUE;
END_IF

IF fbRTrig_ZeroStable_W.Q THEN
	cmd_W 			:= 401;
	writeTrigger_W	:= TRUE;
END_IF

IF fbRTrig_ZeroImm_W.Q THEN
	cmd_W 			:= 404;
	writeTrigger_W	:= TRUE;
END_IF

IF fbRTrig_Clear_W.Q THEN
	cmd_W 			:= 402;
	writeTrigger_W	:= TRUE;
END_IF

IF fbRTrig_PreTare_W.Q THEN
	MB_CmdValue		:= PreTare_value;
	cmd_W 			:= 201;
	writeTrigger_W	:= TRUE;
END_IF

// Deliver the command to the EtherCAT device:
IF writeTrigger_W THEN
	MB_Command		:=	cmd_W;
	MB_CmdValue		:= 	0.0;
	cmdDone			:=	FALSE;
	cmdFailed		:=	FALSE;
	restoreTrigger_W	:=	FALSE;
	writeTrigger_W	:= 	FALSE;
END_IF
// cmdDone status flag will be turned ON if the command resposne is equal to command delivered
// cmdPending status flag is raised when the command response is decimal "2047", the device is trying to execute the command
// cmdFailed status flag will be turned ON if the device finally fails to execute the current command due to motion or out-of-range 
IF MB_Response = UINT_TO_INT(cmd_W) THEN
	cmdDone			:=	TRUE;
	cmdPending		:=	FALSE;
	cmdFailed		:=	FALSE;
	restoreTrigger_W	:=	TRUE;
ELSIF MB_Response = 2047 THEN
	cmdDone			:=	FALSE;
	cmdPending		:=	TRUE;
	cmdFailed		:=	FALSE;
ELSIF MB_Response < 0 THEN
	cmdDone			:=	FALSE;
	cmdPending		:=	FALSE;
	cmdFailed		:=	TRUE;	
	restoreTrigger_W	:=	TRUE;
END_IF
// After scale command is executed/ failed, issue a new command to report the weight data... 
// according to user defined type in "weightCmd"
IF restoreTrigger_W THEN
	MB_Command		:= weightCmd; 
	TareStable_cmd := TareImmediate_cmd := ZeroStable_cmd := ZeroImmediate_cmd := PreTare_cmd := Clear_cmd := FALSE; 
	restoreTrigger_W	:= FALSE;
END_IF

// Continuously updates the device primary status bits
sequence0_W		:=		MB_DeviceStatus.0; 
sequence1_W		:=		MB_DeviceStatus.1;
heartBeat		:=		MB_DeviceStatus.2;
DataOK			:=		MB_DeviceStatus.3;
Smart5_red		:=		MB_DeviceStatus.4;
centerofZero	:=		MB_DeviceStatus.5;
motion			:=		MB_DeviceStatus.6;
netMode			:=		MB_DeviceStatus.7;
Smart5_orange	:=		MB_DeviceStatus.10;
Smart5_yellow	:=		MB_DeviceStatus.11;
Smart5_blue		:=		MB_DeviceStatus.12;

// Updates the real-time and stable weight values continuously
IF (MB_Response <= 3 AND MB_Response >= 0) 
OR (MB_Response <= 7 AND MB_Response >= 5) THEN
	realtimeWeight := MB_MeasuredValue;
	IF NOT motion THEN
		stableWeight := MB_MeasuredValue;
	END_IF
END_IF
END_METHOD

METHOD Set_Zero : BOOL
VAR_INPUT
END_VAR
IF idDevice = 1 THEN
    IND_M_WR_Command := 404;
ELSIF idDevice = 2 THEN
    CMDLaumas := 8;
END_IF
END_METHOD

PROPERTY Status : REAL
GET
IF idDevice = 1 THEN
	status := WORD_TO_REAL(IND_M_RD_Status);
ELSIF idDevice = 2 THEN
	status := DINT_TO_REAL(uStatusLaumas.fReal);
END_IF
END_GET
END_PROPERTY

END_FUNCTION_BLOCK

// ---- POUs/Components/Sim Components/FB_LoadCell_Sim.TcPOU
FUNCTION_BLOCK FB_LoadCell_Sim IMPLEMENTS I_LoadCell
VAR_INPUT
END_VAR
VAR_OUTPUT
END_VAR
VAR
	bEnable : BOOL;
	fValue  : REAL;
	wStatus : WORD;
	// var Sim
	nState  		: INT;
	fSetpoint		: REAL := 1000000;//setpoint feedback speed Loadcell 
	tTimer			: TON; 
	bInit			: BOOL := TRUE;
END_VAR

CASE nState OF
	0: //init
		IF bInit THEN
			fValue := 0;
		END_IF
		nState := nState + 1;
	1://Loadcell Stop
		fValue := 0;
	
	10: // check have cup on loadcell
		IF bHaveLoad THEN
			nState := 20;
		END_IF
	20:
		fValue := fValue + fInvSpeed/fSetpoint;
		IF NOT bHaveLoad THEN
			nState := 10;
		END_IF
END_CASE
//check enable loadcell
IF (nState = 1) AND bEnable THEN
	tTimer(IN := FALSE);
	nState := 10;//Loadcell start
END_IF

PROPERTY fActWeight : REAL
GET
fActWeight := fValue;
END_GET
END_PROPERTY

METHOD NetMode : BOOL
VAR_INPUT
END_VAR
bEnable := true;
END_METHOD

METHOD Set_Zero : BOOL
VAR_INPUT
END_VAR
fValue := 0;
END_METHOD

PROPERTY Status : REAL
GET
Status := WORD_TO_REAL(wStatus);
END_GET
END_PROPERTY

END_FUNCTION_BLOCK

// ---- POUs/Modules/FB_WormWeightModule.TcPOU
FUNCTION_BLOCK FB_WormWeightModule
VAR_INPUT
	nLine							: INT;
	UnitID							: BYTE;
	fFast_Speed_vibrating_funnel	: REAL;
	fSlow_Speed_vibrating_funnel_1	: REAL;
	fSlow_Speed_vibrating_funnel_2	: REAL;
	fDerisedWeight_Worm				: REAL;
	fChangeMode_Worm_1				: REAL;
	fChangeMode_Worm_2				: REAL;
	fMaxWeight_Worm					: REAL;
	fPerStop_Worm					: REAL;
	fTimer_Worm						: REAL;
	fTimer_Alarm_Worm				: REAL;
	fTimer_Error_Worm				: REAL;
	fTimer_Check_Worm				: REAL;
	fTimer_Check_Cylinder			: REAL;
	fDelta_Worm						: REAL;
END_VAR
VAR_OUTPUT
	fProductLog						: ARRAY [1..5] OF REAL;
	bStatus_Worm					: BOOL;
	Time_start						: DT;
	Time_Stop						: DT;
	status							: STRING;
	fweight_iot						: REAL;
END_VAR
VAR 
	// ===== CHILD COMPONENTS ============
	fbInverter 			: FB_Inverter;
	fbCylinder			: FB_Cylinder;
	fbLoadcell			: FB_Loadcell;
	// ===== SIM COMPONENTS ==============
	fbInverterSim		: FB_Inverter_Sim;
	fbCylinderSim		: FB_Cylinder_Sim;
	fbLoadcellSim		: FB_LoadCell_Sim;
	// ===== INTERFACES ==================
	iInverter			: I_Inverter;
	iCylinder			: I_Cylinder;
	iLoadcell			: I_LoadCell;
	// ====== VAR IO =====================
	bCupPresent 	AT %I*	: BOOL;
	bError_Inverter AT %I* 	: BOOL;
	//======= VAR METHOD =================
	nState				: INT;
	nStateWrn			: INT;
	nStateEnable		: INT;
	nStateErr			: INT;
	fbTimer_Err			: TON;
	fbTimer				: TON;
	fbTimer1			: TON;
	fbTimer_Alarm		: TON;	
	fbTimer_Check		: TON;
	fbTimer_Error		: TON;	
	fFastWeight			: REAL;
	fSlowWeight			: REAL;
	fSlowWeight1		: REAL;
	fChangemode_val		: REAL;
	fChangemode_val1	: REAL;
	fLowToleWeight		: REAL;
	fHighToleWeight		: REAL;
	fTareWeight			: REAL;
	bDone				: BOOL;
	p,k					: INT;
	//========= VAR HMI Worm Weight Auto ============
	fFlow_Worm						: REAL;
	fWeight_Worm					: REAL;
	fActDelta_Worm					: REAL;	
	fSpeed_vibrating_funnel_Manual	: REAL := 30;
	fTime							: REAL;
	Error							: BOOL;
	bStatus							: BOOL;
	timestart						: DT;
END_VAR

IF bSimMode THEN
	iInverter	:= fbInverterSim;
	fbInverterSim();
	iCylinder	:= fbCylinderSim;
	fbCylinderSim();
	iLoadcell	:= fbLoadcellSim;
	fbLoadcellSim();
ELSE
	iInverter	:= fbInverter;
	fbInverter(UnitID := UnitID, id := 1);
	iCylinder	:= fbCylinder;
	fbCylinder(id := 1);
	iLoadcell	:= fbLoadcell;
	fbLoadcell(idDevice := nLine,Error=>Error);
END_IF

IF iLoadcell.fActWeight > fMaxWeight_Worm THEN
	IF nLine = 1 THEN
		F_SetError(57,nLine := 1);
	ELSIF nLine = 2 THEN
		F_SetError(59,nLine := 2);
	END_IF
END_IF

IF Error THEN
	IF nLine = 1 THEN
		F_SetError(70,nLine := 1);
	ELSIF nLine = 2 THEN
		F_SetError(72,nLine := 2);
	END_IF
END_IF

IF bIsError_Inverter THEN
	IF nLine = 1 THEN
		F_SetError(9,nLine := 1);
	ELSIF nLine = 2 THEN
		F_SetError(31,nLine := 2);
	END_IF
END_IF

METHOD Auto : BOOL
VAR_INPUT
END_VAR
GetLocalSystemTime(bEnable := 1);
fbTimer(PT 						:= T#100S);
fbTimer_Alarm(PT				:= REAL_TO_TIME(fTimer_Alarm_Worm)*1000);
fbTimer_Check(PT				:= REAL_TO_TIME(fTimer_Check_Cylinder)*1000);
CASE nState OF
	0:// Init Value
		Auto					:= FALSE;
		fbTimer(IN := FALSE);
		fbTimer1(IN := FALSE);
		fbTimer_Alarm(IN := FALSE);
		fbTimer_Check(IN := FALSE);
		fbTimer_Error(IN := FALSE);
		bDone					:= FALSE;	
		nState 					:= 1;
	1:// Init Value
		fFastWeight				:= fFast_Speed_vibrating_funnel;
		fSlowWeight				:= fSlow_Speed_vibrating_funnel_1;
		fSlowWeight1			:= fSlow_Speed_vibrating_funnel_2;
		fChangemode_val			:= fDerisedWeight_Worm*fChangeMode_Worm_1/100;
		fChangemode_val1		:= (fDerisedWeight_Worm - fChangemode_val)*fChangeMode_Worm_2/100 + fChangemode_val;
		fLowToleWeight			:= fDerisedWeight_Worm*(1-(fDelta_Worm/100));
		fHighToleWeight			:= fDerisedWeight_Worm*(1+(fDelta_Worm/100));
		bStatus_Worm			:= FALSE;
		bStatus					:= FALSE;
		fTime					:= 0;
		nState					:= 2;
	2:// Cup detection
		iLoadcell.NetMode();
		IF NOT bIsCupPresent THEN
			fbTimer1(IN := TRUE, PT := REAL_TO_TIME(fTimer_Worm)*1000);
			IF fbTimer1.Q  THEN
				nState	:= 3;
			END_IF
		END_IF
	3:// Tare weight
		timestart := SYSTEMTIME_TO_DT(GetLocalSystemTime.systemTime);
		fbTimer1(IN := FALSE);
		fTareWeight 			:= iLoadcell.fActWeight;
		fWeight_Worm			:= iLoadcell.fActWeight - fTareWeight;
		nState					:= 4;
	4:// Cylinder Retract
		iCylinder.Retract();
		fbTimer_Check(IN := TRUE);
		nState				:= 5;
	5:// Fast Weight
		iCylinder.Retract();
		IF iCylinder.bIsRetract THEN
			fbTimer_Check(IN := FALSE);
		ELSE
			fbTimer_Check(IN := TRUE);
			IF fbTimer_Check.Q THEN
				IF nLine = 1 THEN
					F_SetError(8,nLine := 1);
				ELSIF nLine = 2 THEN
					F_SetError(30,nLine := 2);
				END_IF
			END_IF
		END_IF
		fbTimer_Check(IN := FALSE);
		fbTimer_Alarm(IN := TRUE);
		iInverter.fTargetSpeed 	:= fFastWeight;
		iInverter.Start();
		fWeight_Worm			:= iLoadcell.fActWeight - fTareWeight;
		fbTimer(IN := TRUE);
		fTime := TIME_TO_REAL(fbTimer.ET)/1000;
		fFlow_Worm				:= fWeight_Worm/((TIME_TO_REAL(fbTimer.ET)+0.00001)/1000);
		IF fWeight_Worm >= fChangemode_val THEN
			nState 				:= 6;
		END_IF
	6:// Slow 1 Weight
		iCylinder.Retract();
		iInverter.fTargetSpeed	:= fSlowWeight;
		fbTimer_Alarm(IN := TRUE);
		iInverter.Start();
		fWeight_Worm			:= iLoadcell.fActWeight	- fTareWeight;
		fbTimer(IN := TRUE);
		fTime := TIME_TO_REAL(fbTimer.ET)/1000;
		fFlow_Worm				:= fWeight_Worm/((TIME_TO_REAL(fbTimer.ET)+0.00001)/1000);
		IF fWeight_Worm	>= fChangemode_val1 THEN
			nState				:= 7;
		END_IF
	7:// Slow 2 Weight
		iCylinder.Retract();
		iInverter.fTargetSpeed	:= fSlowWeight1;
		fbTimer_Alarm(IN := TRUE);
		iInverter.Start();
		fWeight_Worm			:= iLoadcell.fActWeight	- fTareWeight;
		fbTimer(IN := TRUE);
		fTime := TIME_TO_REAL(fbTimer.ET)/1000;
		fFlow_Worm				:= fWeight_Worm/((TIME_TO_REAL(fbTimer.ET)+0.00001)/1000);
		IF fWeight_Worm	>= fLowToleWeight*fPerStop_Worm/100 THEN
			nState				:= 8;
		END_IF
	8:// Wait Stable Weight
		iInverter.Stop();
		iCylinder.Extend();
		fbTimer(IN := TRUE);
		fTime := TIME_TO_REAL(fbTimer.ET)/1000;
		fWeight_Worm			:= iLoadcell.fActWeight	- fTareWeight;
		fbTimer1(IN := TRUE, PT := REAL_TO_TIME(fTimer_Check_Worm)*1000);
		IF fbTimer1.Q THEN
			nState				:= 9;
		END_IF
	9:// Check Done
		fbTimer1(IN := FALSE);
		fbTimer_Alarm(IN := TRUE);
		fWeight_Worm			:= iLoadcell.fActWeight	- fTareWeight;
		IF fWeight_Worm < fLowToleWeight THEN
			nState				:= 10;
		ELSIF fWeight_Worm >= fLowToleWeight AND fWeight_Worm <= fHighToleWeight THEN
			nState				:= 11;
		ELSIF fWeight_Worm > fHighToleWeight THEN
			nState				:= 12;	
		END_IF
	10:// No Enough Weight
		fbTimer_Alarm(IN := TRUE);
		iCylinder.Retract();
		fWeight_Worm			:= iLoadcell.fActWeight - fTareWeight;
		iInverter.fTargetSpeed	:= fSlowWeight1;
		iInverter.Start();
		IF fWeight_Worm	>= fLowToleWeight THEN
			nState				:= 8;
		END_IF
	11:// Enough Weight
		iCylinder.Extend();
		fbTimer_Check(IN := TRUE);
		fActDelta_Worm			:= (fWeight_Worm - fDerisedWeight_Worm)/fDerisedWeight_Worm*100;
		fWeight_Worm			:= iLoadcell.fActWeight - fTareWeight;
		fweight_iot				:= iLoadcell.fActWeight - fTareWeight;
		Time_start				:= timestart;
		bStatus_Worm			:= TRUE;
		status					:= 'Pass';
		fbTimer(IN := FALSE);
		fbTimer_Alarm(IN := FALSE);
		bDone					:= TRUE;
		p						:= p + 1;
		nState					:= 13;
	12:// Overweight
		iCylinder.Extend();
		fbTimer_Check(IN := TRUE);
		fActDelta_Worm			:= (fWeight_Worm - fDerisedWeight_Worm)/fDerisedWeight_Worm*100;
		fWeight_Worm			:= iLoadcell.fActWeight - fTareWeight;
		fweight_iot				:= iLoadcell.fActWeight - fTareWeight;
		Time_start				:= timestart;
		bStatus_Worm			:= FALSE;
		status					:= 'Fail';
		fbTimer_Alarm(IN := FALSE);
		fbTimer_Error(IN := FALSE);
		fbTimer(IN := FALSE);
		bDone					:= TRUE;
		p						:= p + 1;
		IF nLine = 1 THEN
			//F_SetWarning(106);
			nState				:= 13;
		ELSIF nLine = 2 THEN
			//F_SetWarning(113);
			nState				:= 13;
		END_IF
	13:// Done
		Time_Stop	:= SYSTEMTIME_TO_DT(GetLocalSystemTime.systemTime);
		bStatus					:= TRUE;
		fbTimer_Check(IN := FALSE);
		IF p > 5 THEN
			p := 5;
		END_IF
		IF bDone THEN
			IF p <> 1 THEN
				FOR k := p TO 2 BY -1 DO
					fProductLog[k] := fProductLog[k-1];
				END_FOR
			END_IF
			fProductLog[1]	:= fWeight_Worm;
			bDone 			:= FALSE;
		END_IF
		Auto					:= TRUE;
		nState					:= 14;
	14:
		nState					:= 0;
END_CASE

//Check Timer WormWeight
CASE nStateWrn OF
	0:
		IF fbTimer_Alarm.Q THEN
			IF nLine = 1 THEN
				F_SetWarning(105,nLine := 1);
			ELSIF nLine = 2 THEN
				F_SetWarning(112,nLine := 2);
			END_IF
			nStateWrn := 1;
		END_IF
	1: 
		IF NOT fbTimer_Alarm.Q THEN
			IF nLine = 1 THEN
					bWrn := FALSE;
			ELSIF nLine = 2 THEN
					bWrn2 := FALSE;
			END_IF
			bSirens := FALSE;
			nStateWrn := 0;
		END_IF
		fbTimer_Error(IN := TRUE, PT := REAL_TO_TIME(fTimer_Error_Worm*1000));
		IF fbTimer_Error.Q THEN
			IF nLine = 1 THEN
				F_SetError(77,nLine := 1);
			ELSIF nLine = 2 THEN
				F_SetError(79,nLine := 2);
			END_IF
			fbTimer_Alarm(IN := FALSE);
			nState := 12;
			nStateWrn := 0;
		END_IF
END_CASE

// Check Fault CupPresent
IF nState > 2 AND nState < 99 THEN
	IF bIsCupPresent THEN
		IF nLine = 1 THEN
			F_SetError(47,nLine := 1);
			nState := 0;
		ELSIF nLine = 2 THEN
			F_SetError(48,nLine := 2);
			nState := 0;
		END_IF
	END_IF
END_IF

// Write ProductLog
END_METHOD

PROPERTY bIsCupPresent : BOOL
GET
bIsCupPresent := bCupPresent;
END_GET
END_PROPERTY

PROPERTY bIsError_Inverter : BOOL
GET
bIsError_Inverter	:= bError_Inverter;
END_GET
END_PROPERTY

METHOD Enable : BOOL
VAR_INPUT
END_VAR
fbTimer_Check(PT := REAL_TO_TIME(fTimer_Check_Cylinder));
CASE nStateEnable OF
	0: //int
		Enable				:= FALSE;
		fbTimer_Check(IN := FALSE);
		nStateEnable 		:= 1;
	1: // Cylinder Extend Block Worm
		iLoadcell.NetMode();
		iCylinder.Extend();
		fbTimer_Check(IN := TRUE);
		IF iCylinder.bIsExtend THEN
			nStateEnable	:= 2;
		ELSIF fbTimer_Check.Q THEN
			nStateEnable	:= 3;
		ELSIF bIsError_Inverter THEN
			nStateEnable	:= 4;
		END_IF
	2: // Enable
		fbTimer_Check(IN := FALSE);
		Enable				:= TRUE;
	3:// Error Cylinder
		IF nLine = 1 THEN
			F_SetError(8,nLine := 1);
			nStateEnable	:= 99;
		ELSIF nLine = 2 THEN
			F_SetError(26,nLine := 2);
			nStateEnable	:= 99;
		END_IF
	4:// Error Inverter
		IF nLine = 1 THEN
			F_SetError(9,nLine := 1);
			nStateEnable	:= 99;
		ELSIF nLine = 2 THEN
			F_SetError(27,nLine := 2);
			nStateEnable	:= 99;
		END_IF
	99:// Error
		iInverter.fTargetSpeed	:= 0;
		iInverter.Stop();
END_CASE
END_METHOD

METHOD Init : BOOL
VAR_INPUT
END_VAR
nState := 0;
nStateEnable := 0;
END_METHOD

METHOD Manual : BOOL
VAR_INPUT
	bUp_vibrating_funnel			: BOOL;
	bDown_vibrating_funnel			: BOOL;
	bZero_Loadcell_Worm				: BOOL;
	bCylinder_Block_Worm_Extend		: BOOL;
	bCylinder_Block_Worm_Retract	: BOOL;
	bMotor_vibrating_funnel			: BOOL;	
END_VAR
IF bUp_vibrating_funnel THEN
	fSpeed_vibrating_funnel_Manual	:= fSpeed_vibrating_funnel_Manual + 0.1;
END_IF

IF bDown_vibrating_funnel THEN
	fSpeed_vibrating_funnel_Manual	:= fSpeed_vibrating_funnel_Manual - 0.1;
END_IF

IF bMotor_vibrating_funnel THEN
	iInverter.Start();
ELSE
	iInverter.Stop();
END_IF

iInverter.fTargetSpeed	:= fSpeed_vibrating_funnel_Manual;

IF bZero_Loadcell_Worm THEN
	iLoadcell.Set_Zero();
ELSE
	iLoadcell.NetMode();
END_IF

fWeight_Worm := iLoadcell.fActWeight;

IF bCylinder_Block_Worm_Extend THEN
	iCylinder.Extend();
	IF NOT iCylinder.bIsRetract THEN
			fbTimer_Check(IN := FALSE);
		ELSE
			fbTimer_Check(IN := TRUE,PT	:= REAL_TO_TIME(fTimer_Check_Cylinder)*1000);
			IF fbTimer_Check.Q THEN
				IF nLine = 1 THEN
					F_SetError(73,nLine := 1);
				ELSIF nLine = 2 THEN
					F_SetError(74,nLine := 2);
				END_IF
			END_IF
	END_IF
END_IF

IF bCylinder_Block_Worm_Retract THEN
	iCylinder.Retract();
		IF iCylinder.bIsRetract THEN
			fbTimer_Check(IN := FALSE);
		ELSE
			fbTimer_Check(IN := TRUE,PT	:= REAL_TO_TIME(fTimer_Check_Cylinder)*1000);
			IF fbTimer_Check.Q THEN
				IF nLine = 1 THEN
					F_SetError(8,nLine := 1);
				ELSIF nLine = 2 THEN
					F_SetError(30,nLine := 2);
				END_IF
			END_IF
	END_IF
END_IF
END_METHOD

METHOD Reset : BOOL
VAR_INPUT
END_VAR
iInverter.Reset();
iCylinder.Extend();
fbTimer(IN := FALSE);			
fbTimer1(IN	:= FALSE);
fbTimer_Alarm(IN := FALSE);
fbTimer_Check(IN := FALSE);
fbTimer_Err(IN := FALSE);
fbTimer_Error(IN := FALSE);
END_METHOD

METHOD SetZero : BOOL
VAR_INPUT
END_VAR
iLoadcell.Set_Zero();
END_METHOD

METHOD Stop : BOOL
VAR_INPUT
END_VAR
iInverter.Stop();
iCylinder.Extend();
fbTimer(IN := FALSE);			
fbTimer1(IN	:= FALSE);
fbTimer_Alarm(IN := FALSE);
fbTimer_Check(IN := FALSE);
fbTimer_Err(IN := FALSE);
fbTimer_Error(IN := FALSE);
END_METHOD

END_FUNCTION_BLOCK

// ---- POUs/Modules/FB_LidSupplyModule.TcPOU
FUNCTION_BLOCK FB_LidSupplyModule
VAR_INPUT
	nLine						: INT;
	timerCylinder_Suction		: REAL := 10;
	timerCheckLidRelease		: REAL := 1;
	timerLidBlow				: REAL := 1;
	timerCheckLidEmpty			: REAL := 1;
	timerCheckLidSuck			: REAL := 1;
	timerCylinder_Stopper		: REAL := 1;
END_VAR
VAR_OUTPUT
END_VAR
VAR
	// ===== CHILD COMPONENTS ======
	fbCylinder_LidStopper		: FB_Cylinder;
	fbCylinder_Suction			: FB_Cylinder;
	fbLidSuctionValve			: FB_SuctionCup;
	fbCupSuctionValve			: FB_SuctionCup;
	// ===== SIM COMPONENTS ======
	fbCylinder_LidStopper_Sim	: FB_Cylinder_Sim;
	fbCylinder_Suction_Sim		: FB_Cylinder_Sim;
	fbLidSuctionValve_Sim		: FB_SuctionCup_Sim;
	fbCupSuctionValve_Sim		: FB_SuctionCup_Sim;
	// ===== INTERFACES ======
	iCylinder_LidStopper		: I_Cylinder;
	iCylinder_Suction			: I_Cylinder;
	iLidSuctionValve			: I_SuctionCup;
	iCupSuctionValve			: I_SuctionCup;
	//===== Var IO ======
	bLidEmpty AT %I*			: BOOL;
	bLidBlow  AT %Q*			: BOOL;
	//===== Var method enable
	nState_Enable				: INT;
	tTimer_Enable				: TON;
	//===== Var method DropLid
	nState_DropLid				: INT;
	tTimer_DropLid				: TON;
	RunDropLid					: BOOL;
	//===== Var method TakeLid
	nState_Check				: INT;
	nState_Siren				: INT;
	nState_TakeLid				: INT;
	tTimer_TakeLid				: TON;
	tTimer_checkLid				: TON;
	//===== var method manual
	tTimer_stoplid				: TON;
	tTimer_Suction				: TON;
	tTimer_Valve				: TON;
	tTimer_Pick					: ton;
END_VAR

IF bSimMode THEN
	iCylinder_LidStopper := fbCylinder_LidStopper_Sim;
	iCylinder_Suction	 := fbCylinder_Suction_Sim;
	iLidSuctionValve	 := fbLidSuctionValve_Sim;
	iCupSuctionValve	 := fbCupSuctionValve_Sim;
	fbCylinder_LidStopper_Sim();
	fbCylinder_Suction_Sim();
	fbLidSuctionValve_Sim();
	fbCupSuctionValve_Sim();
ELSE
	iCylinder_LidStopper := fbCylinder_LidStopper;
	iCylinder_Suction	 := fbCylinder_Suction;
	iLidSuctionValve	 := fbLidSuctionValve;
	iCupSuctionValve	 := fbCupSuctionValve;
	fbCylinder_LidStopper(id := 1);
	fbCylinder_Suction(id := 1);
	fbLidSuctionValve();
	fbCupSuctionValve();
END_IF

METHOD CheckLid : BOOL
VAR_INPUT
END_VAR
IF NOT isLidEmpty THEN
	CASE nState_Check OF
		0:
			IF nLine = 1 THEN
				F_SetWarning(102,nLine := 1);
			ELSIF nLine = 2 THEN
				F_SetWarning(109,nLine := 2);
			END_IF
			nState_Check := 1;
		1:
			tTimer_checkLid(IN := TRUE, PT := REAL_TO_TIME(timerCheckLidEmpty)*1000);
			IF tTimer_checkLid.Q AND NOT RunDropLid THEN
				IF nLine = 1 THEN
					F_SetError(10,nLine := 1);
				ELSIF nLine = 2 THEN
					F_SetError(32,nLine := 2);
				END_IF
			END_IF

	END_CASE
ELSE
	tTimer_checkLid(IN := FALSE);
	nState_Check := 0;
END_IF

CASE nState_Siren OF 
	0:
		IF NOT isLidEmpty THEN
			nState_Siren := 1;
		END_IF
	1:
		IF isLidEmpty THEN
			IF nLine = 1 THEN
				bWrn := FALSE;
			ELSIF nLine = 2 THEN
				bWrn2 := FALSE;
			END_IF
			bSirens := FALSE;
			nState_Siren := 0;
		END_IF
END_CASE
END_METHOD

METHOD DropLid : BOOL
VAR_INPUT
END_VAR
CASE nState_DropLid OF
	0://init
		DropLid := FALSE;
		tTimer_DropLid(IN:= FALSE);
		RunDropLid := FALSE;
		nState_DropLid := 1;
	1://check LidPick
		RunDropLid := TRUE;
		iLidSuctionValve.Suck();
		IF isLidPick THEN
			tTimer_DropLid(IN := FALSE);
			nState_DropLid := 2;
		ELSE
			tTimer_DropLid(IN := TRUE, PT := REAL_TO_TIME(timerCheckLidSuck)*1000);
			IF tTimer_DropLid.Q THEN
				IF nLine = 1 THEN
					F_SetError(49,nLine := 1);
				ELSIF nLine = 2 THEN
					F_SetError(50,nLine := 2);
				END_IF
			END_IF
		END_IF
	2://suck the cup and cylinder_suction retract
		RunDropLid := TRUE;
		iCupSuctionValve.Suck();
		iLidSuctionValve.Suck();
		iCylinder_Suction.Extend();
		IF iCylinder_Suction.bIsExtend THEN
			tTimer_DropLid(IN:= FALSE);
			nState_DropLid := 4;
		ELSE
			tTimer_DropLid(IN:= TRUE,PT := REAL_TO_TIME(timerCylinder_Suction)*1000);
			IF tTimer_DropLid.Q THEN
				IF nLine = 1 THEN
					F_SetError(14,nLine := 1);
				ELSIF nLine = 2 THEN
					F_SetError(36,nLine := 2);
				END_IF
			END_IF
		END_IF
	4://drop Lid
		RunDropLid := TRUE;
		iLidSuctionValve.Release();
		tTimer_DropLid(IN := TRUE, PT := REAL_TO_TIME(timerCheckLidRelease)*1000);
		IF tTimer_DropLid.Q AND NOT isLidPick THEN
			nState_DropLid := 5;
		END_IF
	5:
		RunDropLid := TRUE;
		tTimer_DropLid(IN := FALSE);
		iCylinder_Suction.Retract();
		iCupSuctionValve.Release();
		nState_DropLid := 6;
	6:
		RunDropLid := TRUE;
		IF iCylinder_Suction.bIsRetract THEN
			tTimer_DropLid(IN:= FALSE);
			nState_DropLid := 7;
		ELSE
			tTimer_DropLid(IN:= TRUE,PT := REAL_TO_TIME(timerCylinder_Suction)*1000);
			IF tTimer_DropLid.Q THEN
				IF nLine = 1 THEN
					F_SetError(13,nLine := 1);
				ELSIF nLine = 2 THEN
					F_SetError(35,nLine := 2);
				END_IF
			END_IF
		END_IF
	7://release the cup
		RunDropLid := TRUE;
		tTimer_DropLid(IN := FALSE);
		IF NOT iCupSuctionValve.bIsSuck THEN
			nState_DropLid := 8;
		END_IF
	8://finish
		RunDropLid := FALSE;
		DropLid := TRUE;
		nState_DropLid := 0;
	99://error
		
END_CASE
END_METHOD

METHOD Enable : BOOL
VAR_INPUT
END_VAR
CASE nState_Enable OF
	0:
		Enable := FALSE;
		tTimer_Enable(IN := FALSE);
		nState_Enable := 1;
	1:
		iCylinder_Suction.Retract();
		tTimer_Enable(IN := TRUE,PT := REAL_TO_TIME(timerCylinder_Suction)*1000);
		IF tTimer_Enable.Q THEN
			IF nLine = 1 THEN
				F_SetError(12,nLine := 1);
			ELSIF nLine = 2 THEN
				F_SetError(30,nLine := 2);
			END_IF
		ELSIF iCylinder_Suction.bIsRetract THEN
			tTimer_Enable(IN := FALSE);
			nState_Enable := 2;
		END_IF
	2: 
		iCylinder_LidStopper.Retract();
		tTimer_Enable(IN := TRUE,PT := REAL_TO_TIME(timerCylinder_Stopper)*1000);
		IF tTimer_Enable.Q THEN
			IF nLine = 1 THEN
				F_SetError(13,nLine := 1);
			ELSIF nLine = 2 THEN
				F_SetError(31,nLine := 2);
			END_IF
		ELSIF iCylinder_LidStopper.bIsRetract THEN
			tTimer_Enable(IN := FALSE);
			nState_Enable := 3;
		END_IF
	3:
		Enable := TRUE;
	99://Error
END_CASE
END_METHOD

METHOD Init : BOOL
VAR_INPUT
END_VAR
nState_DropLid := 0;
nState_TakeLid := 0;
nState_Enable  := 0;
END_METHOD

PROPERTY isLidEmpty : BOOL
GET
isLidEmpty := bLidEmpty;
END_GET
END_PROPERTY

PROPERTY isLidPick : BOOL
GET
isLidPick := iLidSuctionValve.bIsSuck;
END_GET
END_PROPERTY

METHOD Manual : BOOL
VAR_INPUT
	bCylinder_LidStopper_extend 	: BOOL;
	bCylinder_LidStopper_retract 	: BOOL;
	bCylinder_Suction_extend		: BOOL;
	bCylinder_Suction_retract		: BOOL;
	bLidSuctionValve				: BOOL;
	bCupSuctionValve				: BOOL;
	bBlowValve						: BOOL;
END_VAR
IF bCylinder_LidStopper_extend THEN
	iCylinder_LidStopper.Extend();
		IF iCylinder_LidStopper.bIsExtend THEN
			tTimer_stoplid(IN := FALSE);
		ELSE
			tTimer_stoplid(IN := TRUE, PT := REAL_TO_TIME(timerCylinder_Stopper)*1000);
			IF tTimer_stoplid.Q THEN
				IF nLine = 1 THEN
					F_SetError(12,nLine := 1);
				ELSIF nLine = 2 THEN
					F_SetError(34,nLine := 2);
				END_IF
			END_IF
		END_IF
END_IF

IF bCylinder_LidStopper_retract THEN
	iCylinder_LidStopper.Retract();
	IF iCylinder_LidStopper.bIsRetract THEN
			tTimer_stoplid(IN := FALSE);
	ELSE
		tTimer_stoplid(IN := TRUE, PT := REAL_TO_TIME(timerCylinder_Stopper)*1000);
		IF tTimer_stoplid.Q THEN
			IF nLine = 1 THEN
				F_SetError(11,nLine := 1);
			ELSIF nLine = 2 THEN
				F_SetError(33,nLine := 2);
			END_IF
		END_IF
	END_IF
END_IF

IF bCylinder_Suction_extend THEN
	iCylinder_Suction.Extend();
	IF iCylinder_Suction.bIsExtend THEN
			tTimer_Suction(IN:= FALSE);
		ELSE
			tTimer_Suction(IN:= TRUE,PT := REAL_TO_TIME(timerCylinder_Suction)*1000);
			IF tTimer_Suction.Q THEN
				IF nLine = 1 THEN
					F_SetError(14,nLine := 1);
				ELSIF nLine = 2 THEN
					F_SetError(36,nLine := 2);
				END_IF
			END_IF
		END_IF
END_IF

IF bCylinder_Suction_retract THEN
	iCylinder_Suction.Retract();
	IF iCylinder_Suction.bIsRetract THEN
			tTimer_Suction(IN := FALSE);
		ELSE
			tTimer_Suction(IN := TRUE, PT := REAL_TO_TIME(timerCylinder_Suction)*1000);
			IF tTimer_Suction.Q THEN
				IF nLine = 1 THEN
					F_SetError(13,nLine := 1);
				ELSIF nLine = 2 THEN
					F_SetError(35,nLine := 2);
				END_IF
			END_IF
		END_IF
END_IF

IF bLidSuctionValve THEN
	iLidSuctionValve.Suck();
	(*IF isLidPick THEN
			tTimer_Valve(IN := FALSE);
		ELSE
			tTimer_Valve(IN := TRUE, PT := REAL_TO_TIME(timerCheckLidSuck)*1000);
			IF tTimer_Valve.Q THEN
				IF nLine = 1 THEN
					F_SetError(49);
				ELSIF nLine = 2 THEN
					F_SetError(50);
				END_IF
			END_IF
		END_IF*)
ELSE
	iLidSuctionValve.Release();
END_IF

IF bCupSuctionValve THEN
	iCupSuctionValve.Suck();
ELSE
	iCupSuctionValve.Release();
END_IF

IF bBlowValve THEN
	bLidBlow := TRUE;
ELSE
	bLidBlow := FALSE;
END_IF
END_METHOD

METHOD Reset : BOOL
VAR_INPUT
END_VAR
tTimer_Enable(IN := FALSE);
tTimer_DropLid(IN := FALSE);
tTimer_TakeLid(IN := FALSE);
tTimer_Suction(IN := FALSE);
tTimer_Pick(IN := FALSE);
iCylinder_Suction.Retract();
END_METHOD

